    |   movel([0.479218, -1.510826, -2.472851, -0.728712, 1.570796, 2.050014],accel_mss,speed_ms,0,blend_radius_m)
    |   movel([0.479090, -1.510544, -2.473106, -0.728739, 1.570796, 2.049886],accel_mss,speed_ms,0,blend_radius_m)
    |   movel([0.478414, -1.510068, -2.473536, -0.728785, 1.570796, 2.049210],accel_mss,speed_ms,0,blend_radius_m)
    |   movel([0.477542, -1.509693, -2.473874, -0.728822, 1.570796, 2.048338],accel_mss,speed_ms,0,blend_radius_m)
    |   movel([0.475558, -1.508835, -2.474647, -0.728907, 1.570796, 2.046354],accel_mss,speed_ms,0,blend_radius_m)
    |   movel([0.473690, -1.507767, -2.475608, -0.729014, 1.570796, 2.044487],accel_mss,speed_ms,0,blend_radius_m)
    |   movel([0.472881, -1.507120, -2.476189, -0.729080, 1.570796, 2.043678],accel_mss,speed_ms,0,blend_radius_m)
    |   movel([0.472200, -1.506379, -2.476853, -0.729157, 1.570796, 2.042997],accel_mss,speed_ms,0,blend_radius_m)
    |   movel([0.471682, -1.505529, -2.477615, -0.729245, 1.570796, 2.042478],accel_mss,speed_ms,0,blend_radius_m)
    |   movel([0.471359, -1.504557, -2.478484, -0.729348, 1.570796, 2.042155],accel_mss,speed_ms,0,blend_radius_m)
    |   movel([0.472548, -1.505063, -2.478031, -0.729294, 1.570796, 2.043345],accel_mss,speed_ms,0,blend_radius_m)
    |   movel([0.473290, -1.505166, -2.477940, -0.729283, 1.570796, 2.044086],accel_mss,speed_ms,0,blend_radius_m)
    |   movel([0.473666, -1.505119, -2.477981, -0.729288, 1.570796, 2.044462],accel_mss,speed_ms,0,blend_radius_m)
    |   movel([0.474036, -1.504983, -2.478103, -0.729303, 1.570796, 2.044833],accel_mss,speed_ms,0,blend_radius_m)
    |   movel([0.474250, -1.504808, -2.478260, -0.729321, 1.570796, 2.045046],accel_mss,speed_ms,0,blend_radius_m)
    |   movel([0.474359, -1.504562, -2.478480, -0.729347, 1.570796, 2.045156],accel_mss,speed_ms,0,blend_radius_m)
    |   movel([0.474320, -1.503904, -2.479067, -0.729418, 1.570796, 2.045117],accel_mss,speed_ms,0,blend_radius_m)
    |   movel([0.474008, -1.503088, -2.479795, -0.729506, 1.570796, 2.044804],accel_mss,speed_ms,0,blend_radius_m)
    |   movel([0.473517, -1.502193, -2.480592, -0.729604, 1.570796, 2.044314],accel_mss,speed_ms,0,blend_radius_m)
    |   movel([0.471613, -1.499414, -2.483059, -0.729917, 1.570796, 2.042409],accel_mss,speed_ms,0,blend_radius_m)
    |   movel([0.471030, -1.498202, -2.484130, -0.730057, 1.570796, 2.041827],accel_mss,speed_ms,0,blend_radius_m)
    |   movel([0.470618, -1.496895, -2.485283, -0.730211, 1.570796, 2.041414],accel_mss,speed_ms,0,blend_radius_m)
    |   movel([0.470446, -1.495493, -2.486518, -0.730379, 1.570796, 2.041242],accel_mss,speed_ms,0,blend_radius_m)
    |   movel([0.470580, -1.493993, -2.487834, -0.730562, 1.570796, 2.041377],accel_mss,speed_ms,0,blend_radius_m)
    |   movel([0.471074, -1.495188, -2.486785, -0.730416, 1.570796, 2.041871],accel_mss,speed_ms,0,blend_radius_m)
    |   movel([0.471484, -1.495742, -2.486298, -0.730349, 1.570796, 2.042280],accel_mss,speed_ms,0,blend_radius_m)
    |   movel([0.472012, -1.496033, -2.486042, -0.730314, 1.570796, 2.042808],accel_mss,speed_ms,0,blend_radius_m)
    |   movel([0.472673, -1.496012, -2.486061, -0.730316, 1.570796, 2.043469],accel_mss,speed_ms,0,blend_radius_m)
    |   movel([0.473211, -1.495731, -2.486308, -0.730350, 1.570796, 2.044007],accel_mss,speed_ms,0,blend_radius_m)
    |   movel([0.473577, -1.495256, -2.486726, -0.730407, 1.570796, 2.044373],accel_mss,speed_ms,0,blend_radius_m)
    |   movel([0.473727, -1.494646, -2.487261, -0.730482, 1.570796, 2.044523],accel_mss,speed_ms,0,blend_radius_m)
    |   movel([0.473997, -1.491440, -2.490067, -0.730882, 1.570796, 2.044794],accel_mss,speed_ms,0,blend_radius_m)
    |   movel([0.474620, -1.488224, -2.492866, -0.731299, 1.570796, 2.045417],accel_mss,speed_ms,0,blend_radius_m)
    |   movel([0.475100, -1.486590, -2.494281, -0.731518, 1.570796, 2.045897],accel_mss,speed_ms,0,blend_radius_m)
    |   movel([0.475711, -1.484927, -2.495718, -0.731745, 1.570796, 2.046507],accel_mss,speed_ms,0,blend_radius_m)
    |   movel([0.476467, -1.483225, -2.497183, -0.731981, 1.570796, 2.047263],accel_mss,speed_ms,0,blend_radius_m)
    |   movel([0.477383, -1.481477, -2.498684, -0.732229, 1.570796, 2.048179],accel_mss,speed_ms,0,blend_radius_m)
    |   speed_ms = 0.005
    |   movel([0.477383, -1.473438, -2.495122, -0.743828, 1.570796, 2.048179],accel_mss,speed_ms,0,blend_radius_m)
    |   speed_ms = 0.040
    |   movel([0.466032, -1.452408, -2.512575, -0.747407, 1.570796, 2.036828],accel_mss,speed_ms,0,blend_radius_m)
    |   speed_ms = 0.005
    |   movel([0.466032, -1.460613, -2.516221, -0.735555, 1.570796, 2.036828],accel_mss,speed_ms,0,blend_radius_m)
    |   speed_ms = 0.025
    |   movel([0.468902, -1.458797, -2.517715, -0.735877, 1.570796, 2.039698],accel_mss,speed_ms,0,blend_radius_m)
    |   movel([0.471734, -1.456911, -2.519262, -0.736216, 1.570796, 2.042530],accel_mss,speed_ms,0,blend_radius_m)
    |   movel([0.477317, -1.452938, -2.522502, -0.736949, 1.570796, 2.048114],accel_mss,speed_ms,0,blend_radius_m)
    |   movel([0.482782, -1.448709, -2.525923, -0.737756, 1.570796, 2.053579],accel_mss,speed_ms,0,blend_radius_m)
    |   movel([0.488116, -1.444241, -2.529509, -0.738639, 1.570796, 2.058913],accel_mss,speed_ms,0,blend_radius_m)
    |   movel([0.493309, -1.439545, -2.533244, -0.739600, 1.570796, 2.064105],accel_mss,speed_ms,0,blend_radius_m)
    |   movel([0.498346, -1.434638, -2.537111, -0.740640, 1.570796, 2.069143],accel_mss,speed_ms,0,blend_radius_m)
    |   movel([0.503214, -1.429536, -2.541092, -0.741760, 1.570796, 2.074011],accel_mss,speed_ms,0,blend_radius_m)
    |   movel([0.507901, -1.424253, -2.545174, -0.742962, 1.570796, 2.078698],accel_mss,speed_ms,0,blend_radius_m)
    |   movel([0.512387, -1.418809, -2.549336, -0.744244, 1.570796, 2.083184],accel_mss,speed_ms,0,blend_radius_m)
    |   movel([0.516658, -1.413219, -2.553563, -0.745607, 1.570796, 2.087454],accel_mss,speed_ms,0,blend_radius_m)
    |   movel([0.520693, -1.407501, -2.557838, -0.747050, 1.570796, 2.091490],accel_mss,speed_ms,0,blend_radius_m)
    |   movel([0.524474, -1.401675, -2.562144, -0.748570, 1.570796, 2.095271],accel_mss,speed_ms,0,blend_radius_m)
    |   movel([0.527986, -1.395759, -2.566466, -0.750164, 1.570796, 2.098783],accel_mss,speed_ms,0,blend_radius_m)
    |   movel([0.531202, -1.389774, -2.570785, -0.751829, 1.570796, 2.101998],accel_mss,speed_ms,0,blend_radius_m)
    |   movel([0.534102, -1.383745, -2.575084, -0.753560, 1.570796, 2.104898],accel_mss,speed_ms,0,blend_radius_m)
    |   movel([0.537945, -1.374648, -2.581470, -0.756271, 1.570796, 2.108741],accel_mss,speed_ms,0,blend_radius_m)
    |   movel([0.538771, -1.373143, -2.582516, -0.756731, 1.570796, 2.109567],accel_mss,speed_ms,0,blend_radius_m)
    |   movel([0.539817, -1.371681, -2.583528, -0.757181, 1.570796, 2.110613],accel_mss,speed_ms,0,blend_radius_m)
    |   movel([0.541538, -1.369792, -2.584831, -0.757767, 1.570796, 2.112334],accel_mss,speed_ms,0,blend_radius_m)
    |   movel([0.543091, -1.368476, -2.585735, -0.758178, 1.570796, 2.113887],accel_mss,speed_ms,0,blend_radius_m)
    |   movel([0.543804, -1.368020, -2.586049, -0.758321, 1.570796, 2.114601],accel_mss,speed_ms,0,blend_radius_m)
    |   movel([0.545113, -1.367469, -2.586426, -0.758494, 1.570796, 2.115909],accel_mss,speed_ms,0,blend_radius_m)
    |   movel([0.545705, -1.367366, -2.586497, -0.758526, 1.570796, 2.116501],accel_mss,speed_ms,0,blend_radius_m)
    |   movel([0.546777, -1.367466, -2.586428, -0.758495, 1.570796, 2.117574],accel_mss,speed_ms,0,blend_radius_m)
    |   movel([0.547701, -1.367929, -2.586111, -0.758349, 1.570796, 2.118497],accel_mss,speed_ms,0,blend_radius_m)
    |   movel([0.548483, -1.368700, -2.585581, -0.758107, 1.570796, 2.119280],accel_mss,speed_ms,0,blend_radius_m)
    |   movel([0.549132, -1.369728, -2.584875, -0.757786, 1.570796, 2.119928],accel_mss,speed_ms,0,blend_radius_m)
    |   movel([0.549655, -1.370952, -2.584031, -0.757406, 1.570796, 2.120452],accel_mss,speed_ms,0,blend_radius_m)
    |   movel([0.550060, -1.372322, -2.583084, -0.756983, 1.570796, 2.120856],accel_mss,speed_ms,0,blend_radius_m)
    |   movel([0.550551, -1.375266, -2.581040, -0.756083, 1.570796, 2.121347],accel_mss,speed_ms,0,blend_radius_m)
    |   movel([0.550668, -1.378132, -2.579039, -0.755219, 1.570796, 2.121464],accel_mss,speed_ms,0,blend_radius_m)
    |   movel([0.550484, -1.380487, -2.577385, -0.754517, 1.570796, 2.121281],accel_mss,speed_ms,0,blend_radius_m)
    |   movel([0.549919, -1.383302, -2.575398, -0.753689, 1.570796, 2.120715],accel_mss,speed_ms,0,blend_radius_m)
    |   movel([0.549155, -1.386148, -2.573377, -0.752864, 1.570796, 2.119951],accel_mss,speed_ms,0,blend_radius_m)
    |   movel([0.547245, -1.391873, -2.569277, -0.751240, 1.570796, 2.118042],accel_mss,speed_ms,0,blend_radius_m)
    |   movel([0.545162, -1.397558, -2.565157, -0.749674, 1.570796, 2.115959],accel_mss,speed_ms,0,blend_radius_m)
    |   movel([0.543302, -1.403099, -2.561096, -0.748194, 1.570796, 2.114098],accel_mss,speed_ms,0,blend_radius_m)
    |   movel([0.541964, -1.407989, -2.557475, -0.746925, 1.570796, 2.112760],accel_mss,speed_ms,0,blend_radius_m)
    |   movel([0.541538, -1.410366, -2.555702, -0.746321, 1.570796, 2.112334],accel_mss,speed_ms,0,blend_radius_m)
    |   movel([0.541409, -1.412652, -2.553988, -0.745748, 1.570796, 2.112205],accel_mss,speed_ms,0,blend_radius_m)
    |   movel([0.541530, -1.413653, -2.553236, -0.745500, 1.570796, 2.112327],accel_mss,speed_ms,0,blend_radius_m)
    |   movel([0.541712, -1.414085, -2.552911, -0.745393, 1.570796, 2.112508],accel_mss,speed_ms,0,blend_radius_m)
    |   movel([0.542014, -1.414430, -2.552651, -0.745308, 1.570796, 2.112811],accel_mss,speed_ms,0,blend_radius_m)
    |   movel([0.542579, -1.414692, -2.552453, -0.745244, 1.570796, 2.113375],accel_mss,speed_ms,0,blend_radius_m)
    |   movel([0.543278, -1.414768, -2.552396, -0.745225, 1.570796, 2.114074],accel_mss,speed_ms,0,blend_radius_m)
    |   movel([0.544866, -1.414552, -2.552559, -0.745278, 1.570796, 2.115662],accel_mss,speed_ms,0,blend_radius_m)
    |   movel([0.546735, -1.414053, -2.552935, -0.745401, 1.570796, 2.117531],accel_mss,speed_ms,0,blend_radius_m)
    |   movel([0.548597, -1.413416, -2.553414, -0.745558, 1.570796, 2.119394],accel_mss,speed_ms,0,blend_radius_m)
    |   movel([0.552310, -1.411832, -2.554605, -0.745953, 1.570796, 2.123106],accel_mss,speed_ms,0,blend_radius_m)
    |   movel([0.559726, -1.408243, -2.557286, -0.746860, 1.570796, 2.130523],accel_mss,speed_ms,0,blend_radius_m)
    |   movel([0.563228, -1.406710, -2.558426, -0.747253, 1.570796, 2.134025],accel_mss,speed_ms,0,blend_radius_m)
    |   movel([0.565185, -1.405992, -2.558959, -0.747439, 1.570796, 2.135981],accel_mss,speed_ms,0,blend_radius_m)
    |   movel([0.567041, -1.405492, -2.559329, -0.747568, 1.570796, 2.137837],accel_mss,speed_ms,0,blend_radius_m)
    |   movel([0.567877, -1.405366, -2.559422, -0.747601, 1.570796, 2.138673],accel_mss,speed_ms,0,blend_radius_m)
    |   movel([0.568623, -1.405347, -2.559436, -0.747606, 1.570796, 2.139419],accel_mss,speed_ms,0,blend_radius_m)
    |   movel([0.569256, -1.405450, -2.559360, -0.747579, 1.570796, 2.140052],accel_mss,speed_ms,0,blend_radius_m)
    |   movel([0.569753, -1.405695, -2.559178, -0.747516, 1.570796, 2.140549],accel_mss,speed_ms,0,blend_radius_m)
    |   movel([0.570094, -1.406095, -2.558882, -0.747412, 1.570796, 2.140890],accel_mss,speed_ms,0,blend_radius_m)
    |   movel([0.570258, -1.406668, -2.558457, -0.747264, 1.570796, 2.141054],accel_mss,speed_ms,0,blend_radius_m)
    |   movel([0.570222, -1.407432, -2.557890, -0.747068, 1.570796, 2.141018],accel_mss,speed_ms,0,blend_radius_m)
    |   movel([0.569963, -1.408401, -2.557168, -0.746820, 1.570796, 2.140760],accel_mss,speed_ms,0,blend_radius_m)
    |   movel([0.569286, -1.410124, -2.555883, -0.746382, 1.570796, 2.140083],accel_mss,speed_ms,0,blend_radius_m)
    |   movel([0.568475, -1.411800, -2.554629, -0.745961, 1.570796, 2.139271],accel_mss,speed_ms,0,blend_radius_m)
    |   movel([0.567540, -1.413425, -2.553408, -0.745556, 1.570796, 2.138336],accel_mss,speed_ms,0,blend_radius_m)
    |   movel([0.566489, -1.415003, -2.552219, -0.745167, 1.570796, 2.137285],accel_mss,speed_ms,0,blend_radius_m)
    |   movel([0.565332, -1.416528, -2.551066, -0.744795, 1.570796, 2.136128],accel_mss,speed_ms,0,blend_radius_m)
    |   movel([0.564077, -1.418002, -2.549949, -0.744438, 1.570796, 2.134873],accel_mss,speed_ms,0,blend_radius_m)
    |   movel([0.562731, -1.419423, -2.548869, -0.744097, 1.570796, 2.133528],accel_mss,speed_ms,0,blend_radius_m)
    |   movel([0.561305, -1.420792, -2.547825, -0.743772, 1.570796, 2.132101],accel_mss,speed_ms,0,blend_radius_m)
    |   movel([0.558245, -1.423366, -2.545855, -0.743168, 1.570796, 2.129041],accel_mss,speed_ms,0,blend_radius_m)
    |   movel([0.554959, -1.425720, -2.544045, -0.742624, 1.570796, 2.125756],accel_mss,speed_ms,0,blend_radius_m)
    |   movel([0.551512, -1.427846, -2.542403, -0.742140, 1.570796, 2.122308],accel_mss,speed_ms,0,blend_radius_m)
    |   movel([0.547970, -1.429739, -2.540935, -0.741715, 1.570796, 2.118766],accel_mss,speed_ms,0,blend_radius_m)
    |   movel([0.539979, -1.433664, -2.537874, -0.740851, 1.570796, 2.110775],accel_mss,speed_ms,0,blend_radius_m)
    |   movel([0.535909, -1.435398, -2.536514, -0.740477, 1.570796, 2.106705],accel_mss,speed_ms,0,blend_radius_m)
    |   movel([0.533914, -1.436111, -2.535954, -0.740324, 1.570796, 2.104710],accel_mss,speed_ms,0,blend_radius_m)
    |   movel([0.531965, -1.436684, -2.535503, -0.740202, 1.570796, 2.102762],accel_mss,speed_ms,0,blend_radius_m)
    |   movel([0.530749, -1.436952, -2.535292, -0.740145, 1.570796, 2.101545],accel_mss,speed_ms,0,blend_radius_m)
    |   movel([0.529585, -1.437111, -2.535167, -0.740111, 1.570796, 2.100382],accel_mss,speed_ms,0,blend_radius_m)
    |   movel([0.528488, -1.437147, -2.535138, -0.740104, 1.570796, 2.099284],accel_mss,speed_ms,0,blend_radius_m)
    |   movel([0.527472, -1.437051, -2.535214, -0.740124, 1.570796, 2.098268],accel_mss,speed_ms,0,blend_radius_m)
    |   movel([0.526552, -1.436813, -2.535401, -0.740174, 1.570796, 2.097349],accel_mss,speed_ms,0,blend_radius_m)
    |   movel([0.525742, -1.436422, -2.535709, -0.740258, 1.570796, 2.096539],accel_mss,speed_ms,0,blend_radius_m)
    |   movel([0.525060, -1.435863, -2.536149, -0.740377, 1.570796, 2.095857],accel_mss,speed_ms,0,blend_radius_m)
    |   movel([0.524520, -1.435125, -2.536729, -0.740535, 1.570796, 2.095316],accel_mss,speed_ms,0,blend_radius_m)
    |   movel([0.524155, -1.434223, -2.537437, -0.740730, 1.570796, 2.094952],accel_mss,speed_ms,0,blend_radius_m)
    |   movel([0.523975, -1.433243, -2.538203, -0.740942, 1.570796, 2.094772],accel_mss,speed_ms,0,blend_radius_m)
    |   movel([0.523875, -1.429029, -2.541486, -0.741874, 1.570796, 2.094671],accel_mss,speed_ms,0,blend_radius_m)
    |   movel([0.523695, -1.428021, -2.542268, -0.742101, 1.570796, 2.094491],accel_mss,speed_ms,0,blend_radius_m)
    |   movel([0.523325, -1.427082, -2.542994, -0.742313, 1.570796, 2.094122],accel_mss,speed_ms,0,blend_radius_m)
    |   movel([0.523071, -1.426813, -2.543202, -0.742374, 1.570796, 2.093867],accel_mss,speed_ms,0,blend_radius_m)
    |   movel([0.522822, -1.426930, -2.543111, -0.742348, 1.570796, 2.093618],accel_mss,speed_ms,0,blend_radius_m)
    |   movel([0.522355, -1.427345, -2.542790, -0.742254, 1.570796, 2.093151],accel_mss,speed_ms,0,blend_radius_m)
    |   movel([0.520874, -1.428916, -2.541574, -0.741899, 1.570796, 2.091670],accel_mss,speed_ms,0,blend_radius_m)
    |   movel([0.516616, -1.433877, -2.537707, -0.740805, 1.570796, 2.087413],accel_mss,speed_ms,0,blend_radius_m)
    |   movel([0.509629, -1.442253, -2.531094, -0.739042, 1.570796, 2.080425],accel_mss,speed_ms,0,blend_radius_m)
    |   movel([0.505584, -1.446410, -2.527772, -0.738207, 1.570796, 2.076380],accel_mss,speed_ms,0,blend_radius_m)
    |   movel([0.501403, -1.450431, -2.524534, -0.737424, 1.570796, 2.072199],accel_mss,speed_ms,0,blend_radius_m)
    |   movel([0.497105, -1.454321, -2.521377, -0.736691, 1.570796, 2.067901],accel_mss,speed_ms,0,blend_radius_m)
    |   movel([0.492719, -1.458086, -2.518299, -0.736004, 1.570796, 2.063515],accel_mss,speed_ms,0,blend_radius_m)
    |   movel([0.487033, -1.462788, -2.514425, -0.735177, 1.570796, 2.057830],accel_mss,speed_ms,0,blend_radius_m)
    |   movel([0.481276, -1.467394, -2.510596, -0.734399, 1.570796, 2.052072],accel_mss,speed_ms,0,blend_radius_m)
    |   movel([0.475444, -1.471860, -2.506851, -0.733677, 1.570796, 2.046241],accel_mss,speed_ms,0,blend_radius_m)
    |   movel([0.469530, -1.476139, -2.503235, -0.733015, 1.570796, 2.040326],accel_mss,speed_ms,0,blend_radius_m)
    |   movel([0.463529, -1.480182, -2.499792, -0.732415, 1.570796, 2.034326],accel_mss,speed_ms,0,blend_radius_m)
    |   movel([0.460496, -1.482104, -2.498146, -0.732139, 1.570796, 2.031292],accel_mss,speed_ms,0,blend_radius_m)
    |   movel([0.457435, -1.483950, -2.496559, -0.731880, 1.570796, 2.028231],accel_mss,speed_ms,0,blend_radius_m)
    |   movel([0.454348, -1.485717, -2.495035, -0.731636, 1.570796, 2.025144],accel_mss,speed_ms,0,blend_radius_m)
    |   movel([0.451235, -1.487398, -2.493582, -0.731409, 1.570796, 2.022032],accel_mss,speed_ms,0,blend_radius_m)
    |   movel([0.448093, -1.488991, -2.492200, -0.731198, 1.570796, 2.018889],accel_mss,speed_ms,0,blend_radius_m)
    |   movel([0.444920, -1.490485, -2.490900, -0.731004, 1.570796, 2.015717],accel_mss,speed_ms,0,blend_radius_m)
    |   movel([0.441121, -1.492138, -2.489458, -0.730793, 1.570796, 2.011917],accel_mss,speed_ms,0,blend_radius_m)
    |   movel([0.439214, -1.492856, -2.488830, -0.730703, 1.570796, 2.010010],accel_mss,speed_ms,0,blend_radius_m)
    |   movel([0.435953, -1.493815, -2.487990, -0.730584, 1.570796, 2.006750],accel_mss,speed_ms,0,blend_radius_m)
    |   movel([0.434355, -1.494140, -2.487706, -0.730544, 1.570796, 2.005151],accel_mss,speed_ms,0,blend_radius_m)
    |   movel([0.432892, -1.494199, -2.487654, -0.730536, 1.570796, 2.003689],accel_mss,speed_ms,0,blend_radius_m)
    |   movel([0.432332, -1.494057, -2.487778, -0.730554, 1.570796, 2.003129],accel_mss,speed_ms,0,blend_radius_m)
    |   movel([0.431947, -1.493762, -2.488037, -0.730590, 1.570796, 2.002743],accel_mss,speed_ms,0,blend_radius_m)
    |   movel([0.433050, -1.492467, -2.489170, -0.730752, 1.570796, 2.003846],accel_mss,speed_ms,0,blend_radius_m)
    |   movel([0.433977, -1.491111, -2.490354, -0.730924, 1.570796, 2.004774],accel_mss,speed_ms,0,blend_radius_m)
    |   movel([0.434304, -1.490444, -2.490936, -0.731009, 1.570796, 2.005100],accel_mss,speed_ms,0,blend_radius_m)
    |   movel([0.434501, -1.489802, -2.491495, -0.731092, 1.570796, 2.005297],accel_mss,speed_ms,0,blend_radius_m)
    |   movel([0.434541, -1.489197, -2.492021, -0.731171, 1.570796, 2.005338],accel_mss,speed_ms,0,blend_radius_m)
    |   movel([0.434390, -1.488645, -2.492501, -0.731244, 1.570796, 2.005186],accel_mss,speed_ms,0,blend_radius_m)
    |   movel([0.433605, -1.487527, -2.493470, -0.731392, 1.570796, 2.004401],accel_mss,speed_ms,0,blend_radius_m)
    |   movel([0.433481, -1.487048, -2.493885, -0.731456, 1.570796, 2.004278],accel_mss,speed_ms,0,blend_radius_m)
    |   movel([0.433504, -1.486523, -2.494339, -0.731527, 1.570796, 2.004300],accel_mss,speed_ms,0,blend_radius_m)
    |   movel([0.433910, -1.485389, -2.495318, -0.731681, 1.570796, 2.004706],accel_mss,speed_ms,0,blend_radius_m)
    |   movel([0.434649, -1.484208, -2.496337, -0.731844, 1.570796, 2.005445],accel_mss,speed_ms,0,blend_radius_m)
    |   movel([0.435548, -1.483069, -2.497317, -0.732003, 1.570796, 2.006344],accel_mss,speed_ms,0,blend_radius_m)
    |   movel([0.438447, -1.479730, -2.500178, -0.732481, 1.570796, 2.009243],accel_mss,speed_ms,0,blend_radius_m)
    |   movel([0.441555, -1.476440, -2.502980, -0.732969, 1.570796, 2.012351],accel_mss,speed_ms,0,blend_radius_m)
    |   movel([0.443204, -1.474853, -2.504325, -0.733211, 1.570796, 2.014000],accel_mss,speed_ms,0,blend_radius_m)
    |   movel([0.444924, -1.473320, -2.505621, -0.733448, 1.570796, 2.015721],accel_mss,speed_ms,0,blend_radius_m)
    |   movel([0.446722, -1.471861, -2.506851, -0.733677, 1.570796, 2.017518],accel_mss,speed_ms,0,blend_radius_m)
    |   movel([0.448605, -1.470491, -2.508003, -0.733895, 1.570796, 2.019402],accel_mss,speed_ms,0,blend_radius_m)
    |   movel([0.450533, -1.469313, -2.508991, -0.734085, 1.570796, 2.021329],accel_mss,speed_ms,0,blend_radius_m)
    |   movel([0.456408, -1.466369, -2.511451, -0.734569, 1.570796, 2.027205],accel_mss,speed_ms,0,blend_radius_m)
    |   movel([0.461233, -1.463560, -2.513785, -0.735044, 1.570796, 2.032030],accel_mss,speed_ms,0,blend_radius_m)
    |   movel([0.466032, -1.460613, -2.516221, -0.735555, 1.570796, 2.036828],accel_mss,speed_ms,0,blend_radius_m)
    |   movel([0.468181, -1.459252, -2.517341, -0.735796, 1.570796, 2.038977],accel_mss,speed_ms,0,blend_radius_m)
    |   speed_ms = 0.005
    |   movel([0.468181, -1.451036, -2.513689, -0.747664, 1.570796, 2.038977],accel_mss,speed_ms,0,blend_radius_m)
    |   speed_ms = 0.040
    |   movel([0.426259, -1.473575, -2.495006, -0.743807, 1.570796, 1.997056],accel_mss,speed_ms,0,blend_radius_m)
    |   speed_ms = 0.005
    |   movel([0.426259, -1.481613, -2.498567, -0.732209, 1.570796, 1.997056],accel_mss,speed_ms,0,blend_radius_m)
    |   speed_ms = 0.025
    |   movel([0.426785, -1.485296, -2.495399, -0.731694, 1.570796, 1.997582],accel_mss,speed_ms,0,blend_radius_m)
    |   movel([0.426943, -1.487302, -2.493665, -0.731422, 1.570796, 1.997739],accel_mss,speed_ms,0,blend_radius_m)
    |   movel([0.426956, -1.489374, -2.491867, -0.731148, 1.570796, 1.997753],accel_mss,speed_ms,0,blend_radius_m)
    |   movel([0.426780, -1.491475, -2.490037, -0.730877, 1.570796, 1.997576],accel_mss,speed_ms,0,blend_radius_m)
    |   movel([0.426361, -1.493570, -2.488205, -0.730614, 1.570796, 1.997157],accel_mss,speed_ms,0,blend_radius_m)
    |   movel([0.425648, -1.495628, -2.486399, -0.730362, 1.570796, 1.996444],accel_mss,speed_ms,0,blend_radius_m)
    |   movel([0.425164, -1.496634, -2.485513, -0.730242, 1.570796, 1.995961],accel_mss,speed_ms,0,blend_radius_m)
    |   movel([0.424590, -1.497615, -2.484648, -0.730126, 1.570796, 1.995386],accel_mss,speed_ms,0,blend_radius_m)
    |   movel([0.424302, -1.496994, -2.485196, -0.730199, 1.570796, 1.995098],accel_mss,speed_ms,0,blend_radius_m)
    |   movel([0.424245, -1.496354, -2.485760, -0.730275, 1.570796, 1.995041],accel_mss,speed_ms,0,blend_radius_m)
    |   movel([0.424185, -1.494900, -2.487039, -0.730451, 1.570796, 1.994982],accel_mss,speed_ms,0,blend_radius_m)
    |   movel([0.423788, -1.493467, -2.488295, -0.730627, 1.570796, 1.994585],accel_mss,speed_ms,0,blend_radius_m)
    |   movel([0.423223, -1.492114, -2.489479, -0.730796, 1.570796, 1.994019],accel_mss,speed_ms,0,blend_radius_m)
    |   movel([0.422503, -1.490843, -2.490588, -0.730958, 1.570796, 1.993300],accel_mss,speed_ms,0,blend_radius_m)
    |   movel([0.421640, -1.489659, -2.491619, -0.731111, 1.570796, 1.992436],accel_mss,speed_ms,0,blend_radius_m)
    |   movel([0.420645, -1.488568, -2.492567, -0.731254, 1.570796, 1.991442],accel_mss,speed_ms,0,blend_radius_m)
    |   movel([0.419531, -1.487577, -2.493427, -0.731385, 1.570796, 1.990327],accel_mss,speed_ms,0,blend_radius_m)
    |   movel([0.418306, -1.486690, -2.494195, -0.731504, 1.570796, 1.989103],accel_mss,speed_ms,0,blend_radius_m)
    |   movel([0.416988, -1.485911, -2.494868, -0.731610, 1.570796, 1.987784],accel_mss,speed_ms,0,blend_radius_m)
    |   movel([0.416041, -1.485484, -2.495237, -0.731668, 1.570796, 1.986838],accel_mss,speed_ms,0,blend_radius_m)
    |   movel([0.415222, -1.485270, -2.495421, -0.731697, 1.570796, 1.986019],accel_mss,speed_ms,0,blend_radius_m)
    |   movel([0.414524, -1.485248, -2.495440, -0.731700, 1.570796, 1.985320],accel_mss,speed_ms,0,blend_radius_m)
    |   movel([0.413938, -1.485397, -2.495312, -0.731680, 1.570796, 1.984734],accel_mss,speed_ms,0,blend_radius_m)
    |   movel([0.413451, -1.485701, -2.495049, -0.731638, 1.570796, 1.984247],accel_mss,speed_ms,0,blend_radius_m)
    |   movel([0.413056, -1.486139, -2.494671, -0.731579, 1.570796, 1.983852],accel_mss,speed_ms,0,blend_radius_m)
    |   movel([0.412740, -1.486691, -2.494194, -0.731504, 1.570796, 1.983536],accel_mss,speed_ms,0,blend_radius_m)
    |   movel([0.412496, -1.487338, -2.493634, -0.731417, 1.570796, 1.983292],accel_mss,speed_ms,0,blend_radius_m)
    |   movel([0.412176, -1.488839, -2.492331, -0.731218, 1.570796, 1.982973],accel_mss,speed_ms,0,blend_radius_m)
    |   movel([0.411827, -1.493652, -2.488133, -0.730604, 1.570796, 1.982623],accel_mss,speed_ms,0,blend_radius_m)
    |   movel([0.411194, -1.492016, -2.489564, -0.730809, 1.570796, 1.981990],accel_mss,speed_ms,0,blend_radius_m)
    |   movel([0.410024, -1.488695, -2.492457, -0.731237, 1.570796, 1.980820],accel_mss,speed_ms,0,blend_radius_m)
    |   movel([0.409157, -1.487197, -2.493756, -0.731436, 1.570796, 1.979953],accel_mss,speed_ms,0,blend_radius_m)
    |   movel([0.407933, -1.485717, -2.495036, -0.731636, 1.570796, 1.978730],accel_mss,speed_ms,0,blend_radius_m)
    |   movel([0.406592, -1.484312, -2.496248, -0.731830, 1.570796, 1.977388],accel_mss,speed_ms,0,blend_radius_m)
    |   movel([0.403823, -1.481556, -2.498615, -0.732217, 1.570796, 1.974619],accel_mss,speed_ms,0,blend_radius_m)
    |   movel([0.402529, -1.480121, -2.499844, -0.732424, 1.570796, 1.973326],accel_mss,speed_ms,0,blend_radius_m)
    |   movel([0.401388, -1.478591, -2.501149, -0.732648, 1.570796, 1.972184],accel_mss,speed_ms,0,blend_radius_m)
    |   movel([0.400466, -1.476926, -2.502567, -0.732896, 1.570796, 1.971262],accel_mss,speed_ms,0,blend_radius_m)
    |   movel([0.399832, -1.475077, -2.504136, -0.733177, 1.570796, 1.970629],accel_mss,speed_ms,0,blend_radius_m)
    |   movel([0.399145, -1.479131, -2.500689, -0.732569, 1.570796, 1.969941],accel_mss,speed_ms,0,blend_radius_m)
    |   movel([0.398904, -1.481187, -2.498932, -0.732270, 1.570796, 1.969701],accel_mss,speed_ms,0,blend_radius_m)
    |   movel([0.398906, -1.483032, -2.497348, -0.732008, 1.570796, 1.969703],accel_mss,speed_ms,0,blend_radius_m)
    |   movel([0.398200, -1.481266, -2.498864, -0.732259, 1.570796, 1.968996],accel_mss,speed_ms,0,blend_radius_m)
    |   movel([0.397271, -1.479624, -2.500269, -0.732497, 1.570796, 1.968068],accel_mss,speed_ms,0,blend_radius_m)
    |   movel([0.395194, -1.476458, -2.502964, -0.732967, 1.570796, 1.965991],accel_mss,speed_ms,0,blend_radius_m)
    |   movel([0.394608, -1.475326, -2.503925, -0.733139, 1.570796, 1.965405],accel_mss,speed_ms,0,blend_radius_m)
    |   movel([0.394185, -1.474140, -2.504928, -0.733321, 1.570796, 1.964981],accel_mss,speed_ms,0,blend_radius_m)
    |   movel([0.393661, -1.471651, -2.507028, -0.733710, 1.570796, 1.964457],accel_mss,speed_ms,0,blend_radius_m)
    |   movel([0.393279, -1.469083, -2.509184, -0.734123, 1.570796, 1.964076],accel_mss,speed_ms,0,blend_radius_m)
    |   movel([0.392690, -1.466536, -2.511311, -0.734542, 1.570796, 1.963486],accel_mss,speed_ms,0,blend_radius_m)
    |   movel([0.392390, -1.465786, -2.511936, -0.734667, 1.570796, 1.963186],accel_mss,speed_ms,0,blend_radius_m)
    |   movel([0.391952, -1.465122, -2.512488, -0.734778, 1.570796, 1.962748],accel_mss,speed_ms,0,blend_radius_m)
    |   movel([0.391326, -1.464651, -2.512880, -0.734858, 1.570796, 1.962122],accel_mss,speed_ms,0,blend_radius_m)
    |   movel([0.390931, -1.464520, -2.512989, -0.734880, 1.570796, 1.961727],accel_mss,speed_ms,0,blend_radius_m)
    |   movel([0.390469, -1.464478, -2.513023, -0.734887, 1.570796, 1.961266],accel_mss,speed_ms,0,blend_radius_m)
    |   movel([0.389918, -1.464541, -2.512972, -0.734877, 1.570796, 1.960714],accel_mss,speed_ms,0,blend_radius_m)
    |   movel([0.389364, -1.464708, -2.512833, -0.734849, 1.570796, 1.960160],accel_mss,speed_ms,0,blend_radius_m)
    |   movel([0.388261, -1.465288, -2.512351, -0.734751, 1.570796, 1.959057],accel_mss,speed_ms,0,blend_radius_m)
    |   movel([0.387204, -1.466087, -2.511686, -0.734616, 1.570796, 1.958001],accel_mss,speed_ms,0,blend_radius_m)
    |   movel([0.386238, -1.466975, -2.510946, -0.734469, 1.570796, 1.957034],accel_mss,speed_ms,0,blend_radius_m)
    |   movel([0.386761, -1.465043, -2.512554, -0.734792, 1.570796, 1.957557],accel_mss,speed_ms,0,blend_radius_m)
    |   movel([0.387114, -1.463166, -2.514112, -0.735111, 1.570796, 1.957911],accel_mss,speed_ms,0,blend_radius_m)
    |   movel([0.387493, -1.459519, -2.517122, -0.735748, 1.570796, 1.958289],accel_mss,speed_ms,0,blend_radius_m)
    |   movel([0.387757, -1.455899, -2.520090, -0.736401, 1.570796, 1.958553],accel_mss,speed_ms,0,blend_radius_m)
    |   movel([0.388297, -1.452167, -2.523127, -0.737094, 1.570796, 1.959094],accel_mss,speed_ms,0,blend_radius_m)
    |   movel([0.388714, -1.450679, -2.524333, -0.737377, 1.570796, 1.959510],accel_mss,speed_ms,0,blend_radius_m)
    |   movel([0.389333, -1.449137, -2.525579, -0.737674, 1.570796, 1.960129],accel_mss,speed_ms,0,blend_radius_m)
    |   movel([0.390119, -1.447559, -2.526849, -0.737981, 1.570796, 1.960915],accel_mss,speed_ms,0,blend_radius_m)
    |   movel([0.391033, -1.445967, -2.528127, -0.738295, 1.570796, 1.961829],accel_mss,speed_ms,0,blend_radius_m)
    |   movel([0.393120, -1.442815, -2.530647, -0.738927, 1.570796, 1.963916],accel_mss,speed_ms,0,blend_radius_m)
    |   movel([0.395304, -1.439843, -2.533008, -0.739538, 1.570796, 1.966100],accel_mss,speed_ms,0,blend_radius_m)
    |   speed_ms = 0.005
    |   movel([0.395304, -1.431474, -2.529275, -0.751640, 1.570796, 1.966100],accel_mss,speed_ms,0,blend_radius_m)
    |   speed_ms = 0.040
    |   # Splitting Linear movement in 2 (instruction 806: MoveL 765)
    |   movel([0.433547, -1.397430, -2.555032, -0.759927, 1.570796, 2.004344],accel_mss,speed_ms,0,blend_radius_m)
    |   movel([0.474434, -1.362082, -2.579990, -0.770317, 1.570796, 2.045231],accel_mss,speed_ms,0,blend_radius_m)
    |   speed_ms = 0.005
    |   movel([0.474434, -1.370965, -2.584022, -0.757402, 1.570796, 2.045231],accel_mss,speed_ms,0,blend_radius_m)
    |   speed_ms = 0.025
    |   movel([0.472989, -1.371456, -2.583683, -0.757250, 1.570796, 2.043785],accel_mss,speed_ms,0,blend_radius_m)
    |   movel([0.472799, -1.371633, -2.583560, -0.757195, 1.570796, 2.043595],accel_mss,speed_ms,0,blend_radius_m)
    |   movel([0.472675, -1.372000, -2.583307, -0.757082, 1.570796, 2.043471],accel_mss,speed_ms,0,blend_radius_m)
    |   movel([0.472603, -1.373262, -2.582433, -0.756694, 1.570796, 2.043400],accel_mss,speed_ms,0,blend_radius_m)
    |   movel([0.473061, -1.377529, -2.579460, -0.755399, 1.570796, 2.043857],accel_mss,speed_ms,0,blend_radius_m)
    |   movel([0.474120, -1.383440, -2.575300, -0.753649, 1.570796, 2.044916],accel_mss,speed_ms,0,blend_radius_m)
    |   movel([0.475543, -1.390187, -2.570489, -0.751713, 1.570796, 2.046339],accel_mss,speed_ms,0,blend_radius_m)
    |   movel([0.478558, -1.403067, -2.561120, -0.748202, 1.570796, 2.049354],accel_mss,speed_ms,0,blend_radius_m)
    |   movel([0.480397, -1.410133, -2.555876, -0.746380, 1.570796, 2.051193],accel_mss,speed_ms,0,blend_radius_m)
    |   movel([0.480639, -1.410710, -2.555445, -0.746234, 1.570796, 2.051436],accel_mss,speed_ms,0,blend_radius_m)
    |   movel([0.481007, -1.411202, -2.555076, -0.746111, 1.570796, 2.051803],accel_mss,speed_ms,0,blend_radius_m)
    |   movel([0.481528, -1.411486, -2.554864, -0.746039, 1.570796, 2.052324],accel_mss,speed_ms,0,blend_radius_m)
    |   movel([0.481855, -1.411515, -2.554842, -0.746032, 1.570796, 2.052651],accel_mss,speed_ms,0,blend_radius_m)
    |   movel([0.482232, -1.411444, -2.554895, -0.746050, 1.570796, 2.053028],accel_mss,speed_ms,0,blend_radius_m)
    |   movel([0.482920, -1.411095, -2.555156, -0.746137, 1.570796, 2.053716],accel_mss,speed_ms,0,blend_radius_m)
    |   movel([0.483556, -1.410598, -2.555529, -0.746263, 1.570796, 2.054352],accel_mss,speed_ms,0,blend_radius_m)
    |   movel([0.486901, -1.407573, -2.557785, -0.747032, 1.570796, 2.057697],accel_mss,speed_ms,0,blend_radius_m)
    |   movel([0.490066, -1.404379, -2.560152, -0.747858, 1.570796, 2.060862],accel_mss,speed_ms,0,blend_radius_m)
    |   movel([0.493048, -1.401044, -2.562608, -0.748737, 1.570796, 2.063844],accel_mss,speed_ms,0,blend_radius_m)
    |   movel([0.495856, -1.397597, -2.565129, -0.749663, 1.570796, 2.066652],accel_mss,speed_ms,0,blend_radius_m)
    |   movel([0.498491, -1.394061, -2.567697, -0.750631, 1.570796, 2.069287],accel_mss,speed_ms,0,blend_radius_m)
    |   movel([0.500957, -1.390465, -2.570289, -0.751635, 1.570796, 2.071754],accel_mss,speed_ms,0,blend_radius_m)
    |   movel([0.503258, -1.386836, -2.572887, -0.752666, 1.570796, 2.074055],accel_mss,speed_ms,0,blend_radius_m)
    |   movel([0.505395, -1.383207, -2.575465, -0.753717, 1.570796, 2.076191],accel_mss,speed_ms,0,blend_radius_m)
    |   movel([0.506270, -1.381540, -2.576643, -0.754206, 1.570796, 2.077066],accel_mss,speed_ms,0,blend_radius_m)
    |   movel([0.506956, -1.379963, -2.577753, -0.754673, 1.570796, 2.077752],accel_mss,speed_ms,0,blend_radius_m)
    |   movel([0.507455, -1.378474, -2.578799, -0.755116, 1.570796, 2.078251],accel_mss,speed_ms,0,blend_radius_m)
    |   movel([0.507775, -1.377073, -2.579780, -0.755537, 1.570796, 2.078572],accel_mss,speed_ms,0,blend_radius_m)
    |   movel([0.507919, -1.375760, -2.580696, -0.755933, 1.570796, 2.078715],accel_mss,speed_ms,0,blend_radius_m)
    |   movel([0.507889, -1.374537, -2.581547, -0.756305, 1.570796, 2.078686],accel_mss,speed_ms,0,blend_radius_m)
    |   movel([0.507696, -1.373399, -2.582338, -0.756652, 1.570796, 2.078492],accel_mss,speed_ms,0,blend_radius_m)
    |   movel([0.507340, -1.372345, -2.583068, -0.756976, 1.570796, 2.078137],accel_mss,speed_ms,0,blend_radius_m)
    |   movel([0.506829, -1.371378, -2.583737, -0.757274, 1.570796, 2.077625],accel_mss,speed_ms,0,blend_radius_m)
    |   movel([0.506167, -1.370497, -2.584345, -0.757547, 1.570796, 2.076963],accel_mss,speed_ms,0,blend_radius_m)
    |   movel([0.505358, -1.369697, -2.584896, -0.757796, 1.570796, 2.076154],accel_mss,speed_ms,0,blend_radius_m)
    |   movel([0.504410, -1.368982, -2.585388, -0.758019, 1.570796, 2.075207],accel_mss,speed_ms,0,blend_radius_m)
    |   movel([0.502113, -1.367799, -2.586200, -0.758390, 1.570796, 2.072910],accel_mss,speed_ms,0,blend_radius_m)
    |   movel([0.499324, -1.366940, -2.586788, -0.758661, 1.570796, 2.070120],accel_mss,speed_ms,0,blend_radius_m)
    |   movel([0.496587, -1.366526, -2.587072, -0.758791, 1.570796, 2.067383],accel_mss,speed_ms,0,blend_radius_m)
    |   movel([0.493687, -1.366467, -2.587112, -0.758810, 1.570796, 2.064483],accel_mss,speed_ms,0,blend_radius_m)
    |   movel([0.490645, -1.366722, -2.586938, -0.758729, 1.570796, 2.061441],accel_mss,speed_ms,0,blend_radius_m)
    |   movel([0.487496, -1.367238, -2.586584, -0.758567, 1.570796, 2.058292],accel_mss,speed_ms,0,blend_radius_m)
    |   movel([0.484273, -1.367969, -2.586083, -0.758337, 1.570796, 2.055069],accel_mss,speed_ms,0,blend_radius_m)
    |   movel([0.481001, -1.368865, -2.585468, -0.758056, 1.570796, 2.051797],accel_mss,speed_ms,0,blend_radius_m)
    |   movel([0.474434, -1.370965, -2.584022, -0.757402, 1.570796, 2.045231],accel_mss,speed_ms,0,blend_radius_m)
    |   movel([0.472989, -1.371456, -2.583683, -0.757250, 1.570796, 2.043785],accel_mss,speed_ms,0,blend_radius_m)
    |   movel([0.472799, -1.371633, -2.583560, -0.757195, 1.570796, 2.043595],accel_mss,speed_ms,0,blend_radius_m)
    |   movel([0.472675, -1.372000, -2.583307, -0.757082, 1.570796, 2.043471],accel_mss,speed_ms,0,blend_radius_m)
    |   movel([0.472651, -1.372400, -2.583030, -0.756959, 1.570796, 2.043448],accel_mss,speed_ms,0,blend_radius_m)
    |   speed_ms = 0.005
    |   movel([0.472651, -1.363527, -2.579005, -0.769857, 1.570796, 2.043448],accel_mss,speed_ms,0,blend_radius_m)
    |   speed_ms = 0.040
    |   movel([0.476821, -1.340541, -2.594336, -0.777512, 1.570796, 2.047618],accel_mss,speed_ms,0,blend_radius_m)
    |   speed_ms = 0.005
    |   movel([0.476821, -1.349572, -2.598463, -0.764353, 1.570796, 2.047618],accel_mss,speed_ms,0,blend_radius_m)
    |   speed_ms = 0.025
    |   movel([0.477677, -1.347959, -2.599526, -0.764904, 1.570796, 2.048473],accel_mss,speed_ms,0,blend_radius_m)
    |   movel([0.478294, -1.346339, -2.600590, -0.765460, 1.570796, 2.049091],accel_mss,speed_ms,0,blend_radius_m)
    |   movel([0.478658, -1.344752, -2.601629, -0.766008, 1.570796, 2.049454],accel_mss,speed_ms,0,blend_radius_m)
    |   movel([0.478760, -1.343233, -2.602620, -0.766537, 1.570796, 2.049556],accel_mss,speed_ms,0,blend_radius_m)
    |   movel([0.478382, -1.339736, -2.604888, -0.767764, 1.570796, 2.049178],accel_mss,speed_ms,0,blend_radius_m)
    |   movel([0.478408, -1.338690, -2.605564, -0.768135, 1.570796, 2.049205],accel_mss,speed_ms,0,blend_radius_m)
    |   movel([0.478593, -1.337680, -2.606215, -0.768494, 1.570796, 2.049389],accel_mss,speed_ms,0,blend_radius_m)
    |   movel([0.478986, -1.336760, -2.606806, -0.768823, 1.570796, 2.049782],accel_mss,speed_ms,0,blend_radius_m)
    |   movel([0.479645, -1.335982, -2.607306, -0.769101, 1.570796, 2.050441],accel_mss,speed_ms,0,blend_radius_m)
    |   movel([0.480625, -1.335334, -2.607721, -0.769334, 1.570796, 2.051421],accel_mss,speed_ms,0,blend_radius_m)
    |   movel([0.481492, -1.335098, -2.607872, -0.769419, 1.570796, 2.052289],accel_mss,speed_ms,0,blend_radius_m)
    |   movel([0.482252, -1.335197, -2.607809, -0.769383, 1.570796, 2.053048],accel_mss,speed_ms,0,blend_radius_m)
    |   movel([0.482905, -1.335552, -2.607581, -0.769256, 1.570796, 2.053701],accel_mss,speed_ms,0,blend_radius_m)
    |   movel([0.483890, -1.336704, -2.606842, -0.768843, 1.570796, 2.054687],accel_mss,speed_ms,0,blend_radius_m)
    |   movel([0.484469, -1.337923, -2.606058, -0.768408, 1.570796, 2.055265],accel_mss,speed_ms,0,blend_radius_m)
    |   movel([0.485197, -1.335855, -2.607387, -0.769147, 1.570796, 2.055994],accel_mss,speed_ms,0,blend_radius_m)
    |   movel([0.485588, -1.333878, -2.608652, -0.769859, 1.570796, 2.056384],accel_mss,speed_ms,0,blend_radius_m)
    |   movel([0.485773, -1.330063, -2.611077, -0.771248, 1.570796, 2.056569],accel_mss,speed_ms,0,blend_radius_m)
    |   movel([0.485880, -1.326195, -2.613517, -0.772677, 1.570796, 2.056677],accel_mss,speed_ms,0,blend_radius_m)
    |   movel([0.486175, -1.324147, -2.614800, -0.773442, 1.570796, 2.056971],accel_mss,speed_ms,0,blend_radius_m)
    |   movel([0.486781, -1.321976, -2.616155, -0.774258, 1.570796, 2.057577],accel_mss,speed_ms,0,blend_radius_m)
    |   movel([0.487335, -1.320582, -2.617021, -0.774786, 1.570796, 2.058131],accel_mss,speed_ms,0,blend_radius_m)
    |   movel([0.487908, -1.319452, -2.617721, -0.775216, 1.570796, 2.058704],accel_mss,speed_ms,0,blend_radius_m)
    |   movel([0.488491, -1.318572, -2.618266, -0.775552, 1.570796, 2.059287],accel_mss,speed_ms,0,blend_radius_m)
    |   movel([0.489074, -1.317931, -2.618661, -0.775797, 1.570796, 2.059870],accel_mss,speed_ms,0,blend_radius_m)
    |   movel([0.489642, -1.317515, -2.618918, -0.775956, 1.570796, 2.060439],accel_mss,speed_ms,0,blend_radius_m)
    |   movel([0.490193, -1.317306, -2.619047, -0.776037, 1.570796, 2.060989],accel_mss,speed_ms,0,blend_radius_m)
    |   movel([0.490709, -1.317289, -2.619057, -0.776043, 1.570796, 2.061506],accel_mss,speed_ms,0,blend_radius_m)
    |   movel([0.491186, -1.317453, -2.618956, -0.775980, 1.570796, 2.061982],accel_mss,speed_ms,0,blend_radius_m)
    |   movel([0.491611, -1.317781, -2.618753, -0.775854, 1.570796, 2.062408],accel_mss,speed_ms,0,blend_radius_m)
    |   movel([0.491974, -1.318257, -2.618460, -0.775672, 1.570796, 2.062770],accel_mss,speed_ms,0,blend_radius_m)
    |   movel([0.492480, -1.319590, -2.617636, -0.775163, 1.570796, 2.063276],accel_mss,speed_ms,0,blend_radius_m)
    |   movel([0.492629, -1.321327, -2.616558, -0.774504, 1.570796, 2.063426],accel_mss,speed_ms,0,blend_radius_m)
    |   movel([0.492348, -1.323346, -2.615301, -0.773742, 1.570796, 2.063144],accel_mss,speed_ms,0,blend_radius_m)
    |   movel([0.493591, -1.321653, -2.616356, -0.774380, 1.570796, 2.064387],accel_mss,speed_ms,0,blend_radius_m)
    |   movel([0.494597, -1.320010, -2.617376, -0.775003, 1.570796, 2.065393],accel_mss,speed_ms,0,blend_radius_m)
    |   movel([0.495417, -1.318404, -2.618369, -0.775616, 1.570796, 2.066213],accel_mss,speed_ms,0,blend_radius_m)
    |   movel([0.497377, -1.313599, -2.621321, -0.777469, 1.570796, 2.068173],accel_mss,speed_ms,0,blend_radius_m)
    |   movel([0.498859, -1.310219, -2.623380, -0.778791, 1.570796, 2.069655],accel_mss,speed_ms,0,blend_radius_m)
    |   movel([0.499616, -1.308827, -2.624223, -0.779339, 1.570796, 2.070412],accel_mss,speed_ms,0,blend_radius_m)
    |   movel([0.500393, -1.307640, -2.624940, -0.779809, 1.570796, 2.071190],accel_mss,speed_ms,0,blend_radius_m)
    |   movel([0.501171, -1.306658, -2.625532, -0.780199, 1.570796, 2.071967],accel_mss,speed_ms,0,blend_radius_m)
    |   movel([0.501934, -1.305878, -2.626001, -0.780510, 1.570796, 2.072731],accel_mss,speed_ms,0,blend_radius_m)
    |   movel([0.502667, -1.305294, -2.626352, -0.780743, 1.570796, 2.073464],accel_mss,speed_ms,0,blend_radius_m)
    |   movel([0.503355, -1.304905, -2.626585, -0.780899, 1.570796, 2.074152],accel_mss,speed_ms,0,blend_radius_m)
    |   movel([0.503982, -1.304707, -2.626704, -0.780978, 1.570796, 2.074779],accel_mss,speed_ms,0,blend_radius_m)
    |   movel([0.504532, -1.304696, -2.626710, -0.780982, 1.570796, 2.075329],accel_mss,speed_ms,0,blend_radius_m)
    |   movel([0.504990, -1.304870, -2.626606, -0.780913, 1.570796, 2.075786],accel_mss,speed_ms,0,blend_radius_m)
    |   movel([0.505340, -1.305221, -2.626395, -0.780772, 1.570796, 2.076136],accel_mss,speed_ms,0,blend_radius_m)
    |   movel([0.505569, -1.305747, -2.626080, -0.780562, 1.570796, 2.076366],accel_mss,speed_ms,0,blend_radius_m)
    |   movel([0.505661, -1.306444, -2.625660, -0.780284, 1.570796, 2.076458],accel_mss,speed_ms,0,blend_radius_m)
    |   movel([0.505600, -1.307307, -2.625140, -0.779941, 1.570796, 2.076396],accel_mss,speed_ms,0,blend_radius_m)
    |   movel([0.505372, -1.308332, -2.624522, -0.779535, 1.570796, 2.076168],accel_mss,speed_ms,0,blend_radius_m)
    |   movel([0.504963, -1.309512, -2.623808, -0.779069, 1.570796, 2.075759],accel_mss,speed_ms,0,blend_radius_m)
    |   movel([0.504361, -1.310843, -2.623001, -0.778545, 1.570796, 2.075158],accel_mss,speed_ms,0,blend_radius_m)
    |   movel([0.505882, -1.309678, -2.623708, -0.779003, 1.570796, 2.076678],accel_mss,speed_ms,0,blend_radius_m)
    |   movel([0.507291, -1.308414, -2.624472, -0.779502, 1.570796, 2.078088],accel_mss,speed_ms,0,blend_radius_m)
    |   movel([0.508613, -1.307071, -2.625283, -0.780035, 1.570796, 2.079409],accel_mss,speed_ms,0,blend_radius_m)
    |   movel([0.509871, -1.305667, -2.626128, -0.780594, 1.570796, 2.080667],accel_mss,speed_ms,0,blend_radius_m)
    |   movel([0.514730, -1.299885, -2.629580, -0.782925, 1.570796, 2.085526],accel_mss,speed_ms,0,blend_radius_m)
    |   movel([0.516568, -1.297775, -2.630828, -0.783786, 1.570796, 2.087364],accel_mss,speed_ms,0,blend_radius_m)
    |   movel([0.518895, -1.295391, -2.632232, -0.784766, 1.570796, 2.089692],accel_mss,speed_ms,0,blend_radius_m)
    |   movel([0.520143, -1.294383, -2.632824, -0.785183, 1.570796, 2.090940],accel_mss,speed_ms,0,blend_radius_m)
    |   movel([0.521391, -1.293655, -2.633250, -0.785484, 1.570796, 2.092187],accel_mss,speed_ms,0,blend_radius_m)
    |   movel([0.522003, -1.293434, -2.633379, -0.785576, 1.570796, 2.092800],accel_mss,speed_ms,0,blend_radius_m)
    |   movel([0.523177, -1.293343, -2.633433, -0.785614, 1.570796, 2.093973],accel_mss,speed_ms,0,blend_radius_m)
    |   movel([0.523727, -1.293507, -2.633336, -0.785546, 1.570796, 2.094523],accel_mss,speed_ms,0,blend_radius_m)
    |   movel([0.524119, -1.293909, -2.633101, -0.785379, 1.570796, 2.094915],accel_mss,speed_ms,0,blend_radius_m)
    |   movel([0.524203, -1.294537, -2.632733, -0.785119, 1.570796, 2.095000],accel_mss,speed_ms,0,blend_radius_m)
    |   movel([0.523804, -1.296075, -2.631830, -0.784484, 1.570796, 2.094600],accel_mss,speed_ms,0,blend_radius_m)
    |   movel([0.522876, -1.298205, -2.630574, -0.783610, 1.570796, 2.093672],accel_mss,speed_ms,0,blend_radius_m)
    |   movel([0.521782, -1.300323, -2.629319, -0.782746, 1.570796, 2.092578],accel_mss,speed_ms,0,blend_radius_m)
    |   movel([0.523955, -1.298870, -2.630181, -0.783338, 1.570796, 2.094752],accel_mss,speed_ms,0,blend_radius_m)
    |   movel([0.526201, -1.297582, -2.630942, -0.783865, 1.570796, 2.096997],accel_mss,speed_ms,0,blend_radius_m)
    |   movel([0.528485, -1.296466, -2.631600, -0.784323, 1.570796, 2.099281],accel_mss,speed_ms,0,blend_radius_m)
    |   movel([0.530768, -1.295526, -2.632153, -0.784710, 1.570796, 2.101564],accel_mss,speed_ms,0,blend_radius_m)
    |   movel([0.535321, -1.293655, -2.633250, -0.785484, 1.570796, 2.106117],accel_mss,speed_ms,0,blend_radius_m)
    |   movel([0.536592, -1.293226, -2.633501, -0.785662, 1.570796, 2.107388],accel_mss,speed_ms,0,blend_radius_m)
    |   movel([0.537753, -1.292944, -2.633665, -0.785779, 1.570796, 2.108550],accel_mss,speed_ms,0,blend_radius_m)
    |   movel([0.538730, -1.292873, -2.633707, -0.785809, 1.570796, 2.109526],accel_mss,speed_ms,0,blend_radius_m)
    |   movel([0.539439, -1.293071, -2.633591, -0.785727, 1.570796, 2.110235],accel_mss,speed_ms,0,blend_radius_m)
    |   movel([0.539796, -1.293629, -2.633265, -0.785495, 1.570796, 2.110592],accel_mss,speed_ms,0,blend_radius_m)
    |   movel([0.539763, -1.294477, -2.632768, -0.785143, 1.570796, 2.110560],accel_mss,speed_ms,0,blend_radius_m)
    |   movel([0.539417, -1.295518, -2.632157, -0.784713, 1.570796, 2.110214],accel_mss,speed_ms,0,blend_radius_m)
    |   movel([0.538829, -1.296650, -2.631491, -0.784247, 1.570796, 2.109626],accel_mss,speed_ms,0,blend_radius_m)
    |   movel([0.538074, -1.297775, -2.630828, -0.783786, 1.570796, 2.108870],accel_mss,speed_ms,0,blend_radius_m)
    |   movel([0.537226, -1.298794, -2.630226, -0.783369, 1.570796, 2.108023],accel_mss,speed_ms,0,blend_radius_m)
    |   movel([0.536357, -1.299608, -2.629743, -0.783037, 1.570796, 2.107154],accel_mss,speed_ms,0,blend_radius_m)
    |   movel([0.535539, -1.300121, -2.629439, -0.782829, 1.570796, 2.106335],accel_mss,speed_ms,0,blend_radius_m)
    |   movel([0.539564, -1.298618, -2.630330, -0.783441, 1.570796, 2.110360],accel_mss,speed_ms,0,blend_radius_m)
    |   movel([0.541559, -1.298052, -2.630664, -0.783672, 1.570796, 2.112356],accel_mss,speed_ms,0,blend_radius_m)
    |   movel([0.543523, -1.297629, -2.630915, -0.783846, 1.570796, 2.114320],accel_mss,speed_ms,0,blend_radius_m)
    |   movel([0.545439, -1.297358, -2.631074, -0.783957, 1.570796, 2.116236],accel_mss,speed_ms,0,blend_radius_m)
    |   movel([0.547294, -1.297255, -2.631135, -0.783999, 1.570796, 2.118090],accel_mss,speed_ms,0,blend_radius_m)
    |   movel([0.549070, -1.297333, -2.631089, -0.783967, 1.570796, 2.119867],accel_mss,speed_ms,0,blend_radius_m)
    |   movel([0.550755, -1.297601, -2.630931, -0.783857, 1.570796, 2.121552],accel_mss,speed_ms,0,blend_radius_m)
    |   movel([0.551714, -1.298079, -2.630649, -0.783661, 1.570796, 2.122511],accel_mss,speed_ms,0,blend_radius_m)
    |   movel([0.552495, -1.298983, -2.630114, -0.783292, 1.570796, 2.123291],accel_mss,speed_ms,0,blend_radius_m)
    |   movel([0.552726, -1.299550, -2.629778, -0.783061, 1.570796, 2.123522],accel_mss,speed_ms,0,blend_radius_m)
    |   movel([0.552803, -1.300169, -2.629411, -0.782809, 1.570796, 2.123599],accel_mss,speed_ms,0,blend_radius_m)
    |   movel([0.552691, -1.300824, -2.629021, -0.782543, 1.570796, 2.123487],accel_mss,speed_ms,0,blend_radius_m)
    |   movel([0.552350, -1.301497, -2.628621, -0.782270, 1.570796, 2.123146],accel_mss,speed_ms,0,blend_radius_m)
    |   movel([0.551814, -1.302079, -2.628275, -0.782035, 1.570796, 2.122610],accel_mss,speed_ms,0,blend_radius_m)
    |   movel([0.551157, -1.302554, -2.627992, -0.781844, 1.570796, 2.121954],accel_mss,speed_ms,0,blend_radius_m)
    |   movel([0.549592, -1.303332, -2.627527, -0.781530, 1.570796, 2.120389],accel_mss,speed_ms,0,blend_radius_m)
    |   movel([0.548029, -1.303757, -2.627273, -0.781359, 1.570796, 2.118825],accel_mss,speed_ms,0,blend_radius_m)
    |   movel([0.546506, -1.303910, -2.627181, -0.781298, 1.570796, 2.117302],accel_mss,speed_ms,0,blend_radius_m)
    |   movel([0.545064, -1.303868, -2.627206, -0.781315, 1.570796, 2.115860],accel_mss,speed_ms,0,blend_radius_m)
    |   movel([0.546236, -1.305031, -2.626509, -0.780848, 1.570796, 2.117032],accel_mss,speed_ms,0,blend_radius_m)
    |   movel([0.547593, -1.306014, -2.625919, -0.780456, 1.570796, 2.118389],accel_mss,speed_ms,0,blend_radius_m)
    |   movel([0.549117, -1.306810, -2.625440, -0.780139, 1.570796, 2.119913],accel_mss,speed_ms,0,blend_radius_m)
    |   movel([0.550792, -1.307414, -2.625076, -0.779899, 1.570796, 2.121588],accel_mss,speed_ms,0,blend_radius_m)
    |   movel([0.552231, -1.307696, -2.624906, -0.779787, 1.570796, 2.123027],accel_mss,speed_ms,0,blend_radius_m)
    |   movel([0.555218, -1.307960, -2.624746, -0.779682, 1.570796, 2.126015],accel_mss,speed_ms,0,blend_radius_m)
    |   movel([0.556664, -1.308230, -2.624584, -0.779575, 1.570796, 2.127460],accel_mss,speed_ms,0,blend_radius_m)
    |   movel([0.558212, -1.308690, -2.624306, -0.779393, 1.570796, 2.129009],accel_mss,speed_ms,0,blend_radius_m)
    |   movel([0.560696, -1.309649, -2.623725, -0.779015, 1.570796, 2.131492],accel_mss,speed_ms,0,blend_radius_m)
    |   movel([0.561790, -1.310255, -2.623358, -0.778776, 1.570796, 2.132586],accel_mss,speed_ms,0,blend_radius_m)
    |   movel([0.562521, -1.310911, -2.622960, -0.778519, 1.570796, 2.133318],accel_mss,speed_ms,0,blend_radius_m)
    |   movel([0.562691, -1.311249, -2.622754, -0.778386, 1.570796, 2.133487],accel_mss,speed_ms,0,blend_radius_m)
    |   movel([0.562694, -1.311591, -2.622546, -0.778252, 1.570796, 2.133490],accel_mss,speed_ms,0,blend_radius_m)
    |   movel([0.562510, -1.311931, -2.622339, -0.778119, 1.570796, 2.133307],accel_mss,speed_ms,0,blend_radius_m)
    |   movel([0.562113, -1.312265, -2.622135, -0.777989, 1.570796, 2.132910],accel_mss,speed_ms,0,blend_radius_m)
    |   movel([0.561025, -1.312830, -2.621791, -0.777768, 1.570796, 2.131822],accel_mss,speed_ms,0,blend_radius_m)
    |   movel([0.559815, -1.313224, -2.621550, -0.777614, 1.570796, 2.130611],accel_mss,speed_ms,0,blend_radius_m)
    |   movel([0.558524, -1.313482, -2.621393, -0.777514, 1.570796, 2.129320],accel_mss,speed_ms,0,blend_radius_m)
    |   movel([0.557205, -1.313629, -2.621303, -0.777457, 1.570796, 2.128001],accel_mss,speed_ms,0,blend_radius_m)
    |   movel([0.554665, -1.313702, -2.621258, -0.777429, 1.570796, 2.125461],accel_mss,speed_ms,0,blend_radius_m)
    |   movel([0.552577, -1.313666, -2.621280, -0.777443, 1.570796, 2.123374],accel_mss,speed_ms,0,blend_radius_m)
    |   movel([0.553095, -1.314568, -2.620728, -0.777093, 1.570796, 2.123892],accel_mss,speed_ms,0,blend_radius_m)
    |   movel([0.553726, -1.315378, -2.620232, -0.776779, 1.570796, 2.124522],accel_mss,speed_ms,0,blend_radius_m)
    |   movel([0.555262, -1.316761, -2.619382, -0.776246, 1.570796, 2.126058],accel_mss,speed_ms,0,blend_radius_m)
    |   movel([0.557070, -1.317890, -2.618687, -0.775813, 1.570796, 2.127867],accel_mss,speed_ms,0,blend_radius_m)
    |   movel([0.559036, -1.318840, -2.618100, -0.775449, 1.570796, 2.129832],accel_mss,speed_ms,0,blend_radius_m)
    |   movel([0.560750, -1.319486, -2.617700, -0.775203, 1.570796, 2.131546],accel_mss,speed_ms,0,blend_radius_m)
    |   movel([0.566077, -1.321158, -2.616663, -0.774568, 1.570796, 2.136873],accel_mss,speed_ms,0,blend_radius_m)
    |   movel([0.566925, -1.321690, -2.616333, -0.774366, 1.570796, 2.137721],accel_mss,speed_ms,0,blend_radius_m)
    |   movel([0.567404, -1.322414, -2.615882, -0.774093, 1.570796, 2.138201],accel_mss,speed_ms,0,blend_radius_m)
    |   movel([0.567376, -1.322780, -2.615654, -0.773955, 1.570796, 2.138172],accel_mss,speed_ms,0,blend_radius_m)
    |   movel([0.567099, -1.323110, -2.615448, -0.773831, 1.570796, 2.137895],accel_mss,speed_ms,0,blend_radius_m)
    |   movel([0.566520, -1.323378, -2.615281, -0.773730, 1.570796, 2.137317],accel_mss,speed_ms,0,blend_radius_m)
    |   movel([0.565588, -1.323554, -2.615171, -0.773664, 1.570796, 2.136384],accel_mss,speed_ms,0,blend_radius_m)
    |   movel([0.564160, -1.323615, -2.615133, -0.773641, 1.570796, 2.134956],accel_mss,speed_ms,0,blend_radius_m)
    |   movel([0.562620, -1.323495, -2.615208, -0.773686, 1.570796, 2.133416],accel_mss,speed_ms,0,blend_radius_m)
    |   movel([0.561231, -1.323153, -2.615421, -0.773815, 1.570796, 2.132027],accel_mss,speed_ms,0,blend_radius_m)
    |   movel([0.560674, -1.322887, -2.615587, -0.773915, 1.570796, 2.131470],accel_mss,speed_ms,0,blend_radius_m)
    |   movel([0.560257, -1.322548, -2.615798, -0.774042, 1.570796, 2.131053],accel_mss,speed_ms,0,blend_radius_m)
    |   movel([0.561241, -1.324942, -2.614303, -0.773144, 1.570796, 2.132038],accel_mss,speed_ms,0,blend_radius_m)
    |   movel([0.562524, -1.327120, -2.612935, -0.772333, 1.570796, 2.133321],accel_mss,speed_ms,0,blend_radius_m)
    |   movel([0.564045, -1.329119, -2.611675, -0.771595, 1.570796, 2.134841],accel_mss,speed_ms,0,blend_radius_m)
    |   movel([0.565745, -1.330982, -2.610496, -0.770912, 1.570796, 2.136541],accel_mss,speed_ms,0,blend_radius_m)
    |   movel([0.569451, -1.334431, -2.608299, -0.769659, 1.570796, 2.140247],accel_mss,speed_ms,0,blend_radius_m)
    |   movel([0.573175, -1.337754, -2.606167, -0.768468, 1.570796, 2.143972],accel_mss,speed_ms,0,blend_radius_m)
    |   movel([0.573691, -1.338478, -2.605701, -0.768210, 1.570796, 2.144487],accel_mss,speed_ms,0,blend_radius_m)
    |   movel([0.573735, -1.338932, -2.605408, -0.768049, 1.570796, 2.144531],accel_mss,speed_ms,0,blend_radius_m)
    |   movel([0.573528, -1.339439, -2.605080, -0.767869, 1.570796, 2.144324],accel_mss,speed_ms,0,blend_radius_m)
    |   movel([0.573099, -1.339888, -2.604790, -0.767711, 1.570796, 2.143896],accel_mss,speed_ms,0,blend_radius_m)
    |   movel([0.571722, -1.340678, -2.604279, -0.767432, 1.570796, 2.142518],accel_mss,speed_ms,0,blend_radius_m)
    |   movel([0.570874, -1.341000, -2.604070, -0.767318, 1.570796, 2.141670],accel_mss,speed_ms,0,blend_radius_m)
    |   movel([0.569183, -1.341339, -2.603851, -0.767199, 1.570796, 2.139979],accel_mss,speed_ms,0,blend_radius_m)
    |   movel([0.567539, -1.341325, -2.603860, -0.767204, 1.570796, 2.138335],accel_mss,speed_ms,0,blend_radius_m)
    |   movel([0.565973, -1.341026, -2.604053, -0.767309, 1.570796, 2.136769],accel_mss,speed_ms,0,blend_radius_m)
    |   movel([0.564526, -1.340506, -2.604390, -0.767492, 1.570796, 2.135323],accel_mss,speed_ms,0,blend_radius_m)
    |   movel([0.563234, -1.339833, -2.604826, -0.767730, 1.570796, 2.134030],accel_mss,speed_ms,0,blend_radius_m)
    |   movel([0.562135, -1.339068, -2.605320, -0.768001, 1.570796, 2.132931],accel_mss,speed_ms,0,blend_radius_m)
    |   movel([0.561270, -1.338276, -2.605831, -0.768282, 1.570796, 2.132067],accel_mss,speed_ms,0,blend_radius_m)
    |   movel([0.561003, -1.338714, -2.605548, -0.768126, 1.570796, 2.131799],accel_mss,speed_ms,0,blend_radius_m)
    |   movel([0.560974, -1.339164, -2.605258, -0.767967, 1.570796, 2.131770],accel_mss,speed_ms,0,blend_radius_m)
    |   movel([0.561152, -1.340097, -2.604655, -0.767637, 1.570796, 2.131948],accel_mss,speed_ms,0,blend_radius_m)
    |   movel([0.561472, -1.340950, -2.604103, -0.767336, 1.570796, 2.132269],accel_mss,speed_ms,0,blend_radius_m)
    |   movel([0.562363, -1.342502, -2.603095, -0.766792, 1.570796, 2.133160],accel_mss,speed_ms,0,blend_radius_m)
    |   movel([0.564091, -1.345024, -2.601451, -0.765914, 1.570796, 2.134887],accel_mss,speed_ms,0,blend_radius_m)
    |   movel([0.565937, -1.347426, -2.599877, -0.765086, 1.570796, 2.136734],accel_mss,speed_ms,0,blend_radius_m)
    |   movel([0.569942, -1.351936, -2.596899, -0.763554, 1.570796, 2.140738],accel_mss,speed_ms,0,blend_radius_m)
    |   movel([0.571032, -1.353216, -2.596049, -0.763124, 1.570796, 2.141829],accel_mss,speed_ms,0,blend_radius_m)
    |   movel([0.571656, -1.354143, -2.595432, -0.762814, 1.570796, 2.142452],accel_mss,speed_ms,0,blend_radius_m)
    |   movel([0.572170, -1.355176, -2.594743, -0.762470, 1.570796, 2.142967],accel_mss,speed_ms,0,blend_radius_m)
    |   movel([0.572449, -1.356251, -2.594024, -0.762114, 1.570796, 2.143245],accel_mss,speed_ms,0,blend_radius_m)
    |   movel([0.572374, -1.357299, -2.593321, -0.761768, 1.570796, 2.143170],accel_mss,speed_ms,0,blend_radius_m)
    |   movel([0.572168, -1.357794, -2.592990, -0.761606, 1.570796, 2.142964],accel_mss,speed_ms,0,blend_radius_m)
    |   movel([0.571829, -1.358259, -2.592677, -0.761453, 1.570796, 2.142626],accel_mss,speed_ms,0,blend_radius_m)
    |   movel([0.571338, -1.358686, -2.592390, -0.761313, 1.570796, 2.142135],accel_mss,speed_ms,0,blend_radius_m)
    |   movel([0.570686, -1.359068, -2.592133, -0.761188, 1.570796, 2.141483],accel_mss,speed_ms,0,blend_radius_m)
    |   movel([0.569974, -1.359179, -2.592058, -0.761152, 1.570796, 2.140771],accel_mss,speed_ms,0,blend_radius_m)
    |   movel([0.569174, -1.359018, -2.592167, -0.761205, 1.570796, 2.139971],accel_mss,speed_ms,0,blend_radius_m)
    |   movel([0.565202, -1.357551, -2.593152, -0.761685, 1.570796, 2.135998],accel_mss,speed_ms,0,blend_radius_m)
    |   movel([0.563995, -1.356820, -2.593642, -0.761926, 1.570796, 2.134792],accel_mss,speed_ms,0,blend_radius_m)
    |   movel([0.563549, -1.356378, -2.593939, -0.762072, 1.570796, 2.134345],accel_mss,speed_ms,0,blend_radius_m)
    |   movel([0.563259, -1.355871, -2.594278, -0.762240, 1.570796, 2.134055],accel_mss,speed_ms,0,blend_radius_m)
    |   movel([0.563894, -1.359000, -2.592178, -0.761210, 1.570796, 2.134690],accel_mss,speed_ms,0,blend_radius_m)
    |   movel([0.564930, -1.361895, -2.590224, -0.760271, 1.570796, 2.135727],accel_mss,speed_ms,0,blend_radius_m)
    |   movel([0.566288, -1.364581, -2.588399, -0.759409, 1.570796, 2.137084],accel_mss,speed_ms,0,blend_radius_m)
    |   movel([0.567890, -1.367082, -2.586691, -0.758616, 1.570796, 2.138687],accel_mss,speed_ms,0,blend_radius_m)
    |   movel([0.569508, -1.368812, -2.585505, -0.758073, 1.570796, 2.140304],accel_mss,speed_ms,0,blend_radius_m)
    |   movel([0.571786, -1.371355, -2.583753, -0.757281, 1.570796, 2.142582],accel_mss,speed_ms,0,blend_radius_m)
    |   movel([0.572698, -1.372726, -2.582804, -0.756859, 1.570796, 2.143494],accel_mss,speed_ms,0,blend_radius_m)
    |   movel([0.573213, -1.374054, -2.581883, -0.756452, 1.570796, 2.144009],accel_mss,speed_ms,0,blend_radius_m)
    |   movel([0.573263, -1.374675, -2.581452, -0.756263, 1.570796, 2.144060],accel_mss,speed_ms,0,blend_radius_m)
    |   movel([0.573144, -1.375252, -2.581050, -0.756087, 1.570796, 2.143941],accel_mss,speed_ms,0,blend_radius_m)
    |   movel([0.572832, -1.375778, -2.580683, -0.755928, 1.570796, 2.143628],accel_mss,speed_ms,0,blend_radius_m)
    |   movel([0.572309, -1.376242, -2.580360, -0.755787, 1.570796, 2.143105],accel_mss,speed_ms,0,blend_radius_m)
    |   movel([0.571702, -1.376584, -2.580121, -0.755684, 1.570796, 2.142498],accel_mss,speed_ms,0,blend_radius_m)
    |   movel([0.571079, -1.376828, -2.579951, -0.755610, 1.570796, 2.141875],accel_mss,speed_ms,0,blend_radius_m)
    |   movel([0.569831, -1.377119, -2.579747, -0.755523, 1.570796, 2.140627],accel_mss,speed_ms,0,blend_radius_m)
    |   movel([0.568531, -1.377283, -2.579632, -0.755473, 1.570796, 2.139327],accel_mss,speed_ms,0,blend_radius_m)
    |   movel([0.566060, -1.377286, -2.579631, -0.755473, 1.570796, 2.136857],accel_mss,speed_ms,0,blend_radius_m)
    |   movel([0.564904, -1.377127, -2.579742, -0.755520, 1.570796, 2.135700],accel_mss,speed_ms,0,blend_radius_m)
    |   movel([0.566200, -1.378941, -2.578471, -0.754977, 1.570796, 2.136997],accel_mss,speed_ms,0,blend_radius_m)
    |   movel([0.567641, -1.380619, -2.577292, -0.754478, 1.570796, 2.138437],accel_mss,speed_ms,0,blend_radius_m)
    |   movel([0.569208, -1.382177, -2.576193, -0.754019, 1.570796, 2.140004],accel_mss,speed_ms,0,blend_radius_m)
    |   movel([0.570887, -1.383627, -2.575167, -0.753594, 1.570796, 2.141683],accel_mss,speed_ms,0,blend_radius_m)
    |   movel([0.574515, -1.386268, -2.573291, -0.752829, 1.570796, 2.145311],accel_mss,speed_ms,0,blend_radius_m)
    |   movel([0.578407, -1.388652, -2.571589, -0.752148, 1.570796, 2.149203],accel_mss,speed_ms,0,blend_radius_m)
    |   movel([0.579346, -1.389428, -2.571034, -0.751928, 1.570796, 2.150143],accel_mss,speed_ms,0,blend_radius_m)
    |   movel([0.579550, -1.389960, -2.570652, -0.751777, 1.570796, 2.150347],accel_mss,speed_ms,0,blend_radius_m)
    |   movel([0.579414, -1.390611, -2.570185, -0.751594, 1.570796, 2.150210],accel_mss,speed_ms,0,blend_radius_m)
    |   movel([0.579137, -1.391041, -2.569875, -0.751473, 1.570796, 2.149933],accel_mss,speed_ms,0,blend_radius_m)
    |   movel([0.578763, -1.391416, -2.569605, -0.751367, 1.570796, 2.149560],accel_mss,speed_ms,0,blend_radius_m)
    |   movel([0.577769, -1.392026, -2.569166, -0.751197, 1.570796, 2.148566],accel_mss,speed_ms,0,blend_radius_m)
    |   movel([0.576546, -1.392460, -2.568853, -0.751076, 1.570796, 2.147343],accel_mss,speed_ms,0,blend_radius_m)
    |   movel([0.575200, -1.392746, -2.568647, -0.750996, 1.570796, 2.145996],accel_mss,speed_ms,0,blend_radius_m)
    |   movel([0.572584, -1.392961, -2.568492, -0.750936, 1.570796, 2.143381],accel_mss,speed_ms,0,blend_radius_m)
    |   movel([0.570809, -1.392845, -2.568576, -0.750969, 1.570796, 2.141605],accel_mss,speed_ms,0,blend_radius_m)
    |   movel([0.571535, -1.393443, -2.568143, -0.750802, 1.570796, 2.142331],accel_mss,speed_ms,0,blend_radius_m)
    |   movel([0.572349, -1.393945, -2.567780, -0.750663, 1.570796, 2.143145],accel_mss,speed_ms,0,blend_radius_m)
    |   movel([0.574202, -1.394682, -2.567247, -0.750460, 1.570796, 2.144998],accel_mss,speed_ms,0,blend_radius_m)
    |   movel([0.576313, -1.395072, -2.566965, -0.750353, 1.570796, 2.147110],accel_mss,speed_ms,0,blend_radius_m)
    |   movel([0.578620, -1.395143, -2.566913, -0.750333, 1.570796, 2.149417],accel_mss,speed_ms,0,blend_radius_m)
    |   movel([0.581071, -1.394908, -2.567083, -0.750398, 1.570796, 2.151867],accel_mss,speed_ms,0,blend_radius_m)
    |   movel([0.583605, -1.394395, -2.567455, -0.750539, 1.570796, 2.154401],accel_mss,speed_ms,0,blend_radius_m)
    |   movel([0.586169, -1.393616, -2.568018, -0.750754, 1.570796, 2.156965],accel_mss,speed_ms,0,blend_radius_m)
    |   movel([0.588706, -1.392596, -2.568755, -0.751038, 1.570796, 2.159502],accel_mss,speed_ms,0,blend_radius_m)
    |   movel([0.589829, -1.392133, -2.569089, -0.751167, 1.570796, 2.160625],accel_mss,speed_ms,0,blend_radius_m)
    |   movel([0.590366, -1.392015, -2.569174, -0.751200, 1.570796, 2.161163],accel_mss,speed_ms,0,blend_radius_m)
    |   movel([0.590849, -1.392039, -2.569157, -0.751193, 1.570796, 2.161645],accel_mss,speed_ms,0,blend_radius_m)
    |   movel([0.591241, -1.392269, -2.568991, -0.751129, 1.570796, 2.162037],accel_mss,speed_ms,0,blend_radius_m)
    |   movel([0.591481, -1.392641, -2.568723, -0.751025, 1.570796, 2.162277],accel_mss,speed_ms,0,blend_radius_m)
    |   movel([0.591567, -1.393380, -2.568189, -0.750820, 1.570796, 2.162364],accel_mss,speed_ms,0,blend_radius_m)
    |   movel([0.591345, -1.394278, -2.567539, -0.750571, 1.570796, 2.162141],accel_mss,speed_ms,0,blend_radius_m)
    |   movel([0.590881, -1.395278, -2.566815, -0.750296, 1.570796, 2.161677],accel_mss,speed_ms,0,blend_radius_m)
    |   movel([0.590241, -1.396332, -2.566049, -0.750007, 1.570796, 2.161037],accel_mss,speed_ms,0,blend_radius_m)
    |   movel([0.588704, -1.398382, -2.564556, -0.749451, 1.570796, 2.159500],accel_mss,speed_ms,0,blend_radius_m)
    |   movel([0.587266, -1.400014, -2.563363, -0.749012, 1.570796, 2.158063],accel_mss,speed_ms,0,blend_radius_m)
    |   movel([0.589604, -1.398798, -2.564252, -0.749339, 1.570796, 2.160401],accel_mss,speed_ms,0,blend_radius_m)
    |   movel([0.591861, -1.397382, -2.565285, -0.749722, 1.570796, 2.162657],accel_mss,speed_ms,0,blend_radius_m)
    |   movel([0.594018, -1.395784, -2.566448, -0.750157, 1.570796, 2.164815],accel_mss,speed_ms,0,blend_radius_m)
    |   movel([0.596054, -1.394033, -2.567717, -0.750639, 1.570796, 2.166851],accel_mss,speed_ms,0,blend_radius_m)
    |   movel([0.597944, -1.392152, -2.569076, -0.751162, 1.570796, 2.168740],accel_mss,speed_ms,0,blend_radius_m)
    |   movel([0.599672, -1.390163, -2.570506, -0.751720, 1.570796, 2.170468],accel_mss,speed_ms,0,blend_radius_m)
    |   movel([0.601208, -1.388096, -2.571987, -0.752306, 1.570796, 2.172005],accel_mss,speed_ms,0,blend_radius_m)
    |   movel([0.602535, -1.385972, -2.573502, -0.752915, 1.570796, 2.173331],accel_mss,speed_ms,0,blend_radius_m)
    |   movel([0.604026, -1.382955, -2.575643, -0.753791, 1.570796, 2.174823],accel_mss,speed_ms,0,blend_radius_m)
    |   movel([0.604912, -1.381390, -2.576749, -0.754250, 1.570796, 2.175709],accel_mss,speed_ms,0,blend_radius_m)
    |   movel([0.605419, -1.380685, -2.577246, -0.754459, 1.570796, 2.176215],accel_mss,speed_ms,0,blend_radius_m)
    |   movel([0.605977, -1.380066, -2.577681, -0.754642, 1.570796, 2.176773],accel_mss,speed_ms,0,blend_radius_m)
    |   movel([0.606991, -1.379225, -2.578272, -0.754892, 1.570796, 2.177787],accel_mss,speed_ms,0,blend_radius_m)
    |   movel([0.607714, -1.378895, -2.578504, -0.754991, 1.570796, 2.178510],accel_mss,speed_ms,0,blend_radius_m)
    |   movel([0.608206, -1.378963, -2.578456, -0.754970, 1.570796, 2.179003],accel_mss,speed_ms,0,blend_radius_m)
    |   movel([0.608528, -1.379314, -2.578209, -0.754866, 1.570796, 2.179324],accel_mss,speed_ms,0,blend_radius_m)
    |   movel([0.609045, -1.380931, -2.577072, -0.754386, 1.570796, 2.179841],accel_mss,speed_ms,0,blend_radius_m)
    |   movel([0.609266, -1.381278, -2.576827, -0.754283, 1.570796, 2.180062],accel_mss,speed_ms,0,blend_radius_m)
    |   movel([0.610734, -1.380000, -2.577727, -0.754662, 1.570796, 2.181531],accel_mss,speed_ms,0,blend_radius_m)
    |   movel([0.612120, -1.378620, -2.578696, -0.755073, 1.570796, 2.182916],accel_mss,speed_ms,0,blend_radius_m)
    |   movel([0.613422, -1.377152, -2.579724, -0.755513, 1.570796, 2.184219],accel_mss,speed_ms,0,blend_radius_m)
    |   movel([0.614645, -1.375605, -2.580804, -0.755980, 1.570796, 2.185441],accel_mss,speed_ms,0,blend_radius_m)
    |   movel([0.615782, -1.373995, -2.581924, -0.756470, 1.570796, 2.186578],accel_mss,speed_ms,0,blend_radius_m)
    |   movel([0.616837, -1.372330, -2.583079, -0.756981, 1.570796, 2.187633],accel_mss,speed_ms,0,blend_radius_m)
    |   movel([0.618706, -1.368889, -2.585451, -0.758048, 1.570796, 2.189502],accel_mss,speed_ms,0,blend_radius_m)
    |   movel([0.620245, -1.365388, -2.587849, -0.759152, 1.570796, 2.191041],accel_mss,speed_ms,0,blend_radius_m)
    |   movel([0.621460, -1.361927, -2.590202, -0.760260, 1.570796, 2.192256],accel_mss,speed_ms,0,blend_radius_m)
    |   movel([0.622342, -1.358612, -2.592439, -0.761337, 1.570796, 2.193139],accel_mss,speed_ms,0,blend_radius_m)
    |   movel([0.622897, -1.355551, -2.594492, -0.762346, 1.570796, 2.193694],accel_mss,speed_ms,0,blend_radius_m)
    |   speed_ms = 0.005
    |   movel([0.622897, -1.346560, -2.590392, -0.775437, 1.570796, 2.193694],accel_mss,speed_ms,0,blend_radius_m)
    |   speed_ms = 0.040
    |   movel([0.610502, -1.345377, -2.591171, -0.775841, 1.570796, 2.181298],accel_mss,speed_ms,0,blend_radius_m)
    |   speed_ms = 0.005
    |   movel([0.610502, -1.354376, -2.595276, -0.762737, 1.570796, 2.181298],accel_mss,speed_ms,0,blend_radius_m)
    |   speed_ms = 0.025
    |   movel([0.610066, -1.353065, -2.596149, -0.763175, 1.570796, 2.180862],accel_mss,speed_ms,0,blend_radius_m)
    |   movel([0.609319, -1.351998, -2.596858, -0.763533, 1.570796, 2.180115],accel_mss,speed_ms,0,blend_radius_m)
    |   movel([0.608310, -1.351150, -2.597420, -0.763819, 1.570796, 2.179106],accel_mss,speed_ms,0,blend_radius_m)
    |   movel([0.607093, -1.350494, -2.597854, -0.764041, 1.570796, 2.177889],accel_mss,speed_ms,0,blend_radius_m)
    |   movel([0.605719, -1.350002, -2.598179, -0.764207, 1.570796, 2.176515],accel_mss,speed_ms,0,blend_radius_m)
    |   movel([0.604238, -1.349647, -2.598414, -0.764328, 1.570796, 2.175034],accel_mss,speed_ms,0,blend_radius_m)
    |   movel([0.601170, -1.349236, -2.598685, -0.764468, 1.570796, 2.171966],accel_mss,speed_ms,0,blend_radius_m)
    |   speed_ms = 0.005
    |   movel([0.601170, -1.340202, -2.594557, -0.777630, 1.570796, 2.171966],accel_mss,speed_ms,0,blend_radius_m)
    |   speed_ms = 0.040
    |   movel([0.605361, -1.340299, -2.594494, -0.777596, 1.570796, 2.176157],accel_mss,speed_ms,0,blend_radius_m)
    |   speed_ms = 0.005
    |   movel([0.605361, -1.349332, -2.598622, -0.764435, 1.570796, 2.176157],accel_mss,speed_ms,0,blend_radius_m)
    |   speed_ms = 0.025
    |   movel([0.606903, -1.347649, -2.599730, -0.765010, 1.570796, 2.177699],accel_mss,speed_ms,0,blend_radius_m)
    |   movel([0.608271, -1.345949, -2.600846, -0.765595, 1.570796, 2.179067],accel_mss,speed_ms,0,blend_radius_m)
    |   movel([0.609470, -1.344228, -2.601971, -0.766190, 1.570796, 2.180267],accel_mss,speed_ms,0,blend_radius_m)
    |   movel([0.610511, -1.342486, -2.603105, -0.766797, 1.570796, 2.181308],accel_mss,speed_ms,0,blend_radius_m)
    |   movel([0.611405, -1.340723, -2.604250, -0.767416, 1.570796, 2.182201],accel_mss,speed_ms,0,blend_radius_m)
    |   movel([0.612159, -1.338937, -2.605405, -0.768047, 1.570796, 2.182955],accel_mss,speed_ms,0,blend_radius_m)
    |   movel([0.612782, -1.337127, -2.606570, -0.768691, 1.570796, 2.183579],accel_mss,speed_ms,0,blend_radius_m)
    |   movel([0.613285, -1.335293, -2.607747, -0.769349, 1.570796, 2.184082],accel_mss,speed_ms,0,blend_radius_m)
    |   movel([0.614347, -1.329963, -2.611141, -0.771285, 1.570796, 2.185143],accel_mss,speed_ms,0,blend_radius_m)
    |   movel([0.614957, -1.327383, -2.612770, -0.772236, 1.570796, 2.185753],accel_mss,speed_ms,0,blend_radius_m)
    |   movel([0.615950, -1.324518, -2.614568, -0.773302, 1.570796, 2.186746],accel_mss,speed_ms,0,blend_radius_m)
    |   movel([0.617539, -1.320905, -2.616820, -0.774663, 1.570796, 2.188336],accel_mss,speed_ms,0,blend_radius_m)
    |   movel([0.619412, -1.317279, -2.619063, -0.776047, 1.570796, 2.190208],accel_mss,speed_ms,0,blend_radius_m)
    |   movel([0.621631, -1.313688, -2.621267, -0.777434, 1.570796, 2.192427],accel_mss,speed_ms,0,blend_radius_m)
    |   movel([0.622890, -1.311921, -2.622345, -0.778123, 1.570796, 2.193686],accel_mss,speed_ms,0,blend_radius_m)
    |   movel([0.624259, -1.310184, -2.623400, -0.778804, 1.570796, 2.195056],accel_mss,speed_ms,0,blend_radius_m)
    |   movel([0.626580, -1.307633, -2.624944, -0.779812, 1.570796, 2.197376],accel_mss,speed_ms,0,blend_radius_m)
    |   movel([0.629067, -1.305352, -2.626317, -0.780720, 1.570796, 2.199863],accel_mss,speed_ms,0,blend_radius_m)
    |   movel([0.631695, -1.303353, -2.627514, -0.781522, 1.570796, 2.202491],accel_mss,speed_ms,0,blend_radius_m)
    |   movel([0.634436, -1.301648, -2.628531, -0.782209, 1.570796, 2.205232],accel_mss,speed_ms,0,blend_radius_m)
    |   movel([0.637256, -1.300253, -2.629361, -0.782775, 1.570796, 2.208052],accel_mss,speed_ms,0,blend_radius_m)
    |   movel([0.640128, -1.299181, -2.629997, -0.783211, 1.570796, 2.210925],accel_mss,speed_ms,0,blend_radius_m)
    |   movel([0.643026, -1.298442, -2.630434, -0.783513, 1.570796, 2.213822],accel_mss,speed_ms,0,blend_radius_m)
    |   movel([0.645914, -1.298048, -2.630667, -0.783674, 1.570796, 2.216711],accel_mss,speed_ms,0,blend_radius_m)
    |   movel([0.648024, -1.297993, -2.630700, -0.783697, 1.570796, 2.218820],accel_mss,speed_ms,0,blend_radius_m)
    |   movel([0.650051, -1.298145, -2.630609, -0.783634, 1.570796, 2.220848],accel_mss,speed_ms,0,blend_radius_m)
    |   movel([0.651979, -1.298499, -2.630400, -0.783490, 1.570796, 2.222776],accel_mss,speed_ms,0,blend_radius_m)
    |   movel([0.653801, -1.299040, -2.630080, -0.783269, 1.570796, 2.224597],accel_mss,speed_ms,0,blend_radius_m)
    |   movel([0.655496, -1.299767, -2.629649, -0.782973, 1.570796, 2.226292],accel_mss,speed_ms,0,blend_radius_m)
    |   movel([0.657053, -1.300666, -2.629116, -0.782607, 1.570796, 2.227849],accel_mss,speed_ms,0,blend_radius_m)
    |   movel([0.658458, -1.301728, -2.628484, -0.782177, 1.570796, 2.229254],accel_mss,speed_ms,0,blend_radius_m)
    |   movel([0.659698, -1.302944, -2.627759, -0.781686, 1.570796, 2.230494],accel_mss,speed_ms,0,blend_radius_m)
    |   movel([0.660758, -1.304304, -2.626945, -0.781140, 1.570796, 2.231554],accel_mss,speed_ms,0,blend_radius_m)
    |   movel([0.661630, -1.305798, -2.626049, -0.780542, 1.570796, 2.232426],accel_mss,speed_ms,0,blend_radius_m)
    |   movel([0.662298, -1.307417, -2.625075, -0.779898, 1.570796, 2.233095],accel_mss,speed_ms,0,blend_radius_m)
    |   movel([0.662753, -1.309151, -2.624027, -0.779211, 1.570796, 2.233549],accel_mss,speed_ms,0,blend_radius_m)
    |   movel([0.662982, -1.310989, -2.622912, -0.778488, 1.570796, 2.233779],accel_mss,speed_ms,0,blend_radius_m)
    |   movel([0.662971, -1.312923, -2.621734, -0.777732, 1.570796, 2.233767],accel_mss,speed_ms,0,blend_radius_m)
    |   movel([0.662713, -1.314939, -2.620501, -0.776949, 1.570796, 2.233509],accel_mss,speed_ms,0,blend_radius_m)
    |   movel([0.662194, -1.317034, -2.619214, -0.776141, 1.570796, 2.232990],accel_mss,speed_ms,0,blend_radius_m)
    |   movel([0.661222, -1.319798, -2.617507, -0.775084, 1.570796, 2.232018],accel_mss,speed_ms,0,blend_radius_m)
    |   movel([0.660038, -1.322566, -2.615787, -0.774036, 1.570796, 2.230834],accel_mss,speed_ms,0,blend_radius_m)
    |   movel([0.658688, -1.325329, -2.614061, -0.773000, 1.570796, 2.229485],accel_mss,speed_ms,0,blend_radius_m)
    |   movel([0.657229, -1.328072, -2.612336, -0.771981, 1.570796, 2.228025],accel_mss,speed_ms,0,blend_radius_m)
    |   movel([0.653850, -1.333959, -2.608600, -0.769830, 1.570796, 2.224647],accel_mss,speed_ms,0,blend_radius_m)
    |   movel([0.650268, -1.339770, -2.604866, -0.767752, 1.570796, 2.221064],accel_mss,speed_ms,0,blend_radius_m)
    |   movel([0.646532, -1.345512, -2.601132, -0.765745, 1.570796, 2.217329],accel_mss,speed_ms,0,blend_radius_m)
    |   movel([0.642701, -1.351180, -2.597400, -0.763809, 1.570796, 2.213498],accel_mss,speed_ms,0,blend_radius_m)
    |   movel([0.627487, -1.373203, -2.582474, -0.756712, 1.570796, 2.198284],accel_mss,speed_ms,0,blend_radius_m)
    |   movel([0.620438, -1.383934, -2.574950, -0.753505, 1.570796, 2.191235],accel_mss,speed_ms,0,blend_radius_m)
    |   movel([0.617107, -1.389270, -2.571147, -0.751972, 1.570796, 2.187903],accel_mss,speed_ms,0,blend_radius_m)
    |   movel([0.613962, -1.394580, -2.567321, -0.750488, 1.570796, 2.184759],accel_mss,speed_ms,0,blend_radius_m)
    |   movel([0.611040, -1.399864, -2.563473, -0.749052, 1.570796, 2.181837],accel_mss,speed_ms,0,blend_radius_m)
    |   movel([0.608382, -1.405119, -2.559605, -0.747665, 1.570796, 2.179179],accel_mss,speed_ms,0,blend_radius_m)
    |   movel([0.606022, -1.410342, -2.555720, -0.746327, 1.570796, 2.176819],accel_mss,speed_ms,0,blend_radius_m)
    |   movel([0.604002, -1.415533, -2.551818, -0.745037, 1.570796, 2.174798],accel_mss,speed_ms,0,blend_radius_m)
    |   movel([0.603351, -1.417541, -2.550299, -0.744549, 1.570796, 2.174148],accel_mss,speed_ms,0,blend_radius_m)
    |   movel([0.602934, -1.419507, -2.548805, -0.744078, 1.570796, 2.173730],accel_mss,speed_ms,0,blend_radius_m)
    |   movel([0.602913, -1.421316, -2.547425, -0.743648, 1.570796, 2.173709],accel_mss,speed_ms,0,blend_radius_m)
    |   movel([0.603103, -1.422127, -2.546805, -0.743457, 1.570796, 2.173899],accel_mss,speed_ms,0,blend_radius_m)
    |   movel([0.603457, -1.422856, -2.546246, -0.743287, 1.570796, 2.174253],accel_mss,speed_ms,0,blend_radius_m)
    |   speed_ms = 0.005
    |   movel([0.603457, -1.414356, -2.542440, -0.755592, 1.570796, 2.174253],accel_mss,speed_ms,0,blend_radius_m)
    |   speed_ms = 0.040
    |   movel([0.603863, -1.383508, -2.565076, -0.763806, 1.570796, 2.174659],accel_mss,speed_ms,0,blend_radius_m)
    |   speed_ms = 0.005
    |   movel([0.603863, -1.392238, -2.569014, -0.751138, 1.570796, 2.174659],accel_mss,speed_ms,0,blend_radius_m)
    |   speed_ms = 0.025
    |   movel([0.603127, -1.392685, -2.568691, -0.751013, 1.570796, 2.173924],accel_mss,speed_ms,0,blend_radius_m)
    |   movel([0.602452, -1.393269, -2.568270, -0.750851, 1.570796, 2.173248],accel_mss,speed_ms,0,blend_radius_m)
    |   movel([0.601838, -1.393967, -2.567765, -0.750657, 1.570796, 2.172634],accel_mss,speed_ms,0,blend_radius_m)
    |   movel([0.601271, -1.394766, -2.567186, -0.750437, 1.570796, 2.172067],accel_mss,speed_ms,0,blend_radius_m)
    |   movel([0.600275, -1.396590, -2.565862, -0.749937, 1.570796, 2.171071],accel_mss,speed_ms,0,blend_radius_m)
    |   movel([0.599419, -1.398598, -2.564398, -0.749393, 1.570796, 2.170215],accel_mss,speed_ms,0,blend_radius_m)
    |   movel([0.597252, -1.404343, -2.560179, -0.747867, 1.570796, 2.168049],accel_mss,speed_ms,0,blend_radius_m)
    |   movel([0.596512, -1.405711, -2.559167, -0.747512, 1.570796, 2.167309],accel_mss,speed_ms,0,blend_radius_m)
    |   movel([0.596041, -1.406232, -2.558780, -0.747377, 1.570796, 2.166837],accel_mss,speed_ms,0,blend_radius_m)
    |   movel([0.595523, -1.406503, -2.558579, -0.747307, 1.570796, 2.166319],accel_mss,speed_ms,0,blend_radius_m)
    |   movel([0.595134, -1.406544, -2.558549, -0.747296, 1.570796, 2.165930],accel_mss,speed_ms,0,blend_radius_m)
    |   movel([0.594860, -1.406384, -2.558668, -0.747337, 1.570796, 2.165656],accel_mss,speed_ms,0,blend_radius_m)
    |   movel([0.594686, -1.406051, -2.558915, -0.747423, 1.570796, 2.165483],accel_mss,speed_ms,0,blend_radius_m)
    |   movel([0.594599, -1.404973, -2.559712, -0.747703, 1.570796, 2.165395],accel_mss,speed_ms,0,blend_radius_m)
    |   movel([0.594773, -1.403540, -2.560772, -0.748078, 1.570796, 2.165569],accel_mss,speed_ms,0,blend_radius_m)
    |   movel([0.595504, -1.400500, -2.563007, -0.748882, 1.570796, 2.166300],accel_mss,speed_ms,0,blend_radius_m)
    |   movel([0.596090, -1.398758, -2.564281, -0.749349, 1.570796, 2.166886],accel_mss,speed_ms,0,blend_radius_m)
    |   movel([0.594372, -1.400820, -2.562772, -0.748797, 1.570796, 2.165169],accel_mss,speed_ms,0,blend_radius_m)
    |   movel([0.592915, -1.402977, -2.561186, -0.748226, 1.570796, 2.163712],accel_mss,speed_ms,0,blend_radius_m)
    |   movel([0.591689, -1.405202, -2.559544, -0.747644, 1.570796, 2.162485],accel_mss,speed_ms,0,blend_radius_m)
    |   movel([0.590673, -1.407457, -2.557871, -0.747061, 1.570796, 2.161469],accel_mss,speed_ms,0,blend_radius_m)
    |   movel([0.589835, -1.409717, -2.556187, -0.746485, 1.570796, 2.160631],accel_mss,speed_ms,0,blend_radius_m)
    |   movel([0.589156, -1.411947, -2.554518, -0.745924, 1.570796, 2.159953],accel_mss,speed_ms,0,blend_radius_m)
    |   movel([0.588161, -1.416200, -2.551315, -0.744875, 1.570796, 2.158957],accel_mss,speed_ms,0,blend_radius_m)
    |   movel([0.587799, -1.417025, -2.550690, -0.744674, 1.570796, 2.158595],accel_mss,speed_ms,0,blend_radius_m)
    |   movel([0.587486, -1.417336, -2.550454, -0.744599, 1.570796, 2.158282],accel_mss,speed_ms,0,blend_radius_m)
    |   movel([0.587116, -1.417448, -2.550369, -0.744572, 1.570796, 2.157912],accel_mss,speed_ms,0,blend_radius_m)
    |   movel([0.586787, -1.417282, -2.550495, -0.744612, 1.570796, 2.157583],accel_mss,speed_ms,0,blend_radius_m)
    |   movel([0.586231, -1.416604, -2.551009, -0.744776, 1.570796, 2.157027],accel_mss,speed_ms,0,blend_radius_m)
    |   movel([0.585878, -1.415801, -2.551616, -0.744972, 1.570796, 2.156674],accel_mss,speed_ms,0,blend_radius_m)
    |   movel([0.585699, -1.414896, -2.552299, -0.745193, 1.570796, 2.156495],accel_mss,speed_ms,0,blend_radius_m)
    |   movel([0.585677, -1.413906, -2.553045, -0.745437, 1.570796, 2.156473],accel_mss,speed_ms,0,blend_radius_m)
    |   movel([0.586007, -1.411768, -2.554652, -0.745969, 1.570796, 2.156803],accel_mss,speed_ms,0,blend_radius_m)
    |   movel([0.586683, -1.409559, -2.556305, -0.746525, 1.570796, 2.157480],accel_mss,speed_ms,0,blend_radius_m)
    |   movel([0.584424, -1.413569, -2.553299, -0.745521, 1.570796, 2.155220],accel_mss,speed_ms,0,blend_radius_m)
    |   movel([0.583494, -1.415563, -2.551796, -0.745030, 1.570796, 2.154290],accel_mss,speed_ms,0,blend_radius_m)
    |   movel([0.582805, -1.417562, -2.550283, -0.744544, 1.570796, 2.153601],accel_mss,speed_ms,0,blend_radius_m)
    |   movel([0.582532, -1.419260, -2.548993, -0.744136, 1.570796, 2.153328],accel_mss,speed_ms,0,blend_radius_m)
    |   movel([0.582490, -1.422386, -2.546606, -0.743397, 1.570796, 2.153286],accel_mss,speed_ms,0,blend_radius_m)
    |   movel([0.582207, -1.424030, -2.545345, -0.743014, 1.570796, 2.153004],accel_mss,speed_ms,0,blend_radius_m)
    |   movel([0.582086, -1.424369, -2.545085, -0.742935, 1.570796, 2.152883],accel_mss,speed_ms,0,blend_radius_m)
    |   movel([0.581854, -1.424681, -2.544845, -0.742863, 1.570796, 2.152650],accel_mss,speed_ms,0,blend_radius_m)
    |   movel([0.581493, -1.424854, -2.544712, -0.742823, 1.570796, 2.152289],accel_mss,speed_ms,0,blend_radius_m)
    |   movel([0.581028, -1.424852, -2.544713, -0.742824, 1.570796, 2.151824],accel_mss,speed_ms,0,blend_radius_m)
    |   movel([0.579948, -1.424500, -2.544984, -0.742905, 1.570796, 2.150744],accel_mss,speed_ms,0,blend_radius_m)
    |   movel([0.578329, -1.423569, -2.545699, -0.743121, 1.570796, 2.149126],accel_mss,speed_ms,0,blend_radius_m)
    |   movel([0.577960, -1.424862, -2.544706, -0.742821, 1.570796, 2.148756],accel_mss,speed_ms,0,blend_radius_m)
    |   movel([0.577645, -1.426357, -2.543554, -0.742478, 1.570796, 2.148441],accel_mss,speed_ms,0,blend_radius_m)
    |   movel([0.577453, -1.428005, -2.542280, -0.742104, 1.570796, 2.148249],accel_mss,speed_ms,0,blend_radius_m)
    |   movel([0.577452, -1.429760, -2.540919, -0.741710, 1.570796, 2.148248],accel_mss,speed_ms,0,blend_radius_m)
    |   movel([0.578459, -1.432834, -2.538523, -0.741032, 1.570796, 2.149255],accel_mss,speed_ms,0,blend_radius_m)
    |   movel([0.578981, -1.434604, -2.537138, -0.740648, 1.570796, 2.149777],accel_mss,speed_ms,0,blend_radius_m)
    |   movel([0.579054, -1.435266, -2.536618, -0.740505, 1.570796, 2.149851],accel_mss,speed_ms,0,blend_radius_m)
    |   movel([0.578930, -1.435676, -2.536296, -0.740417, 1.570796, 2.149726],accel_mss,speed_ms,0,blend_radius_m)
    |   movel([0.578610, -1.435930, -2.536097, -0.740363, 1.570796, 2.149406],accel_mss,speed_ms,0,blend_radius_m)
    |   movel([0.578244, -1.436091, -2.535970, -0.740328, 1.570796, 2.149040],accel_mss,speed_ms,0,blend_radius_m)
    |   movel([0.577528, -1.436139, -2.535932, -0.740318, 1.570796, 2.148324],accel_mss,speed_ms,0,blend_radius_m)
    |   movel([0.577053, -1.435949, -2.536081, -0.740359, 1.570796, 2.147850],accel_mss,speed_ms,0,blend_radius_m)
    |   movel([0.576639, -1.435645, -2.536321, -0.740424, 1.570796, 2.147435],accel_mss,speed_ms,0,blend_radius_m)
    |   movel([0.575903, -1.434975, -2.536847, -0.740568, 1.570796, 2.146700],accel_mss,speed_ms,0,blend_radius_m)
    |   movel([0.575457, -1.436740, -2.535459, -0.740190, 1.570796, 2.146253],accel_mss,speed_ms,0,blend_radius_m)
    |   movel([0.575152, -1.438476, -2.534090, -0.739824, 1.570796, 2.145948],accel_mss,speed_ms,0,blend_radius_m)
    |   movel([0.574992, -1.440172, -2.532747, -0.739470, 1.570796, 2.145788],accel_mss,speed_ms,0,blend_radius_m)
    |   movel([0.574969, -1.441823, -2.531436, -0.739130, 1.570796, 2.145765],accel_mss,speed_ms,0,blend_radius_m)
    |   movel([0.575168, -1.443368, -2.530206, -0.738815, 1.570796, 2.145964],accel_mss,speed_ms,0,blend_radius_m)
    |   movel([0.575609, -1.444795, -2.529066, -0.738528, 1.570796, 2.146405],accel_mss,speed_ms,0,blend_radius_m)
    |   movel([0.576832, -1.447452, -2.526935, -0.738002, 1.570796, 2.147628],accel_mss,speed_ms,0,blend_radius_m)
    |   movel([0.577055, -1.448296, -2.526256, -0.737837, 1.570796, 2.147851],accel_mss,speed_ms,0,blend_radius_m)
    |   movel([0.576965, -1.448753, -2.525888, -0.737748, 1.570796, 2.147761],accel_mss,speed_ms,0,blend_radius_m)
    |   movel([0.576654, -1.449187, -2.525538, -0.737664, 1.570796, 2.147450],accel_mss,speed_ms,0,blend_radius_m)
    |   movel([0.576237, -1.449464, -2.525315, -0.737610, 1.570796, 2.147034],accel_mss,speed_ms,0,blend_radius_m)
    |   movel([0.575782, -1.449602, -2.525204, -0.737584, 1.570796, 2.146578],accel_mss,speed_ms,0,blend_radius_m)
    |   movel([0.574884, -1.449595, -2.525209, -0.737585, 1.570796, 2.145680],accel_mss,speed_ms,0,blend_radius_m)
    |   movel([0.573821, -1.449344, -2.525411, -0.737633, 1.570796, 2.144617],accel_mss,speed_ms,0,blend_radius_m)
    |   movel([0.572869, -1.448961, -2.525721, -0.737708, 1.570796, 2.143665],accel_mss,speed_ms,0,blend_radius_m)
    |   movel([0.572013, -1.448465, -2.526120, -0.737804, 1.570796, 2.142809],accel_mss,speed_ms,0,blend_radius_m)
    |   movel([0.571243, -1.447873, -2.526597, -0.737919, 1.570796, 2.142039],accel_mss,speed_ms,0,blend_radius_m)
    |   movel([0.571156, -1.449345, -2.525410, -0.737633, 1.570796, 2.141952],accel_mss,speed_ms,0,blend_radius_m)
    |   movel([0.571249, -1.450744, -2.524280, -0.737365, 1.570796, 2.142045],accel_mss,speed_ms,0,blend_radius_m)
    |   movel([0.571531, -1.452045, -2.523227, -0.737117, 1.570796, 2.142327],accel_mss,speed_ms,0,blend_radius_m)
    |   movel([0.572008, -1.453226, -2.522267, -0.736895, 1.570796, 2.142804],accel_mss,speed_ms,0,blend_radius_m)
    |   movel([0.572690, -1.454268, -2.521420, -0.736701, 1.570796, 2.143486],accel_mss,speed_ms,0,blend_radius_m)
    |   movel([0.573586, -1.455151, -2.520700, -0.736538, 1.570796, 2.144382],accel_mss,speed_ms,0,blend_radius_m)
    |   movel([0.574704, -1.455850, -2.520130, -0.736410, 1.570796, 2.145500],accel_mss,speed_ms,0,blend_radius_m)
    |   movel([0.576054, -1.456348, -2.519722, -0.736318, 1.570796, 2.146850],accel_mss,speed_ms,0,blend_radius_m)
    |   speed_ms = 0.005
    |   movel([0.576054, -1.448109, -2.516058, -0.748222, 1.570796, 2.146850],accel_mss,speed_ms,0,blend_radius_m)
    |   speed_ms = 0.040
    |   movel([0.585604, -1.442287, -2.520731, -0.749370, 1.570796, 2.156400],accel_mss,speed_ms,0,blend_radius_m)
    |   speed_ms = 0.005
    |   movel([0.585604, -1.450572, -2.524420, -0.737398, 1.570796, 2.156400],accel_mss,speed_ms,0,blend_radius_m)
    |   speed_ms = 0.025
    |   movel([0.583814, -1.448240, -2.526302, -0.737848, 1.570796, 2.154611],accel_mss,speed_ms,0,blend_radius_m)
    |   movel([0.583126, -1.447097, -2.527220, -0.738071, 1.570796, 2.153922],accel_mss,speed_ms,0,blend_radius_m)
    |   movel([0.582592, -1.445916, -2.528168, -0.738305, 1.570796, 2.153389],accel_mss,speed_ms,0,blend_radius_m)
    |   movel([0.582226, -1.444649, -2.529183, -0.738557, 1.570796, 2.153022],accel_mss,speed_ms,0,blend_radius_m)
    |   movel([0.582039, -1.443255, -2.530296, -0.738838, 1.570796, 2.152835],accel_mss,speed_ms,0,blend_radius_m)
    |   movel([0.582043, -1.441690, -2.531542, -0.739157, 1.570796, 2.152839],accel_mss,speed_ms,0,blend_radius_m)
    |   movel([0.582253, -1.439911, -2.532954, -0.739524, 1.570796, 2.153050],accel_mss,speed_ms,0,blend_radius_m)
    |   movel([0.583077, -1.436109, -2.535956, -0.740325, 1.570796, 2.153873],accel_mss,speed_ms,0,blend_radius_m)
    |   movel([0.584263, -1.432233, -2.538993, -0.741163, 1.570796, 2.155059],accel_mss,speed_ms,0,blend_radius_m)
    |   movel([0.585769, -1.428306, -2.542047, -0.742036, 1.570796, 2.156566],accel_mss,speed_ms,0,blend_radius_m)
    |   movel([0.587548, -1.424355, -2.545096, -0.742938, 1.570796, 2.158344],accel_mss,speed_ms,0,blend_radius_m)
    |   movel([0.589196, -1.421115, -2.547579, -0.743696, 1.570796, 2.159993],accel_mss,speed_ms,0,blend_radius_m)
    |   movel([0.590996, -1.417874, -2.550046, -0.744469, 1.570796, 2.161792],accel_mss,speed_ms,0,blend_radius_m)
    |   movel([0.594940, -1.411377, -2.554946, -0.746067, 1.570796, 2.165736],accel_mss,speed_ms,0,blend_radius_m)
    |   movel([0.609438, -1.388730, -2.571533, -0.752125, 1.570796, 2.180234],accel_mss,speed_ms,0,blend_radius_m)
    |   movel([0.612520, -1.383868, -2.574997, -0.753524, 1.570796, 2.183317],accel_mss,speed_ms,0,blend_radius_m)
    |   movel([0.615548, -1.378943, -2.578470, -0.754976, 1.570796, 2.186344],accel_mss,speed_ms,0,blend_radius_m)
    |   movel([0.618446, -1.373967, -2.581944, -0.756479, 1.570796, 2.189243],accel_mss,speed_ms,0,blend_radius_m)
    |   movel([0.621146, -1.368941, -2.585416, -0.758032, 1.570796, 2.191942],accel_mss,speed_ms,0,blend_radius_m)
    |   movel([0.623574, -1.363874, -2.588880, -0.759635, 1.570796, 2.194371],accel_mss,speed_ms,0,blend_radius_m)
    |   movel([0.625657, -1.358775, -2.592330, -0.761284, 1.570796, 2.196453],accel_mss,speed_ms,0,blend_radius_m)
    |   movel([0.626927, -1.355048, -2.594828, -0.762513, 1.570796, 2.197723],accel_mss,speed_ms,0,blend_radius_m)
    |   movel([0.628014, -1.351222, -2.597372, -0.763795, 1.570796, 2.198811],accel_mss,speed_ms,0,blend_radius_m)
    |   movel([0.628873, -1.347360, -2.599920, -0.765109, 1.570796, 2.199669],accel_mss,speed_ms,0,blend_radius_m)
    |   movel([0.629455, -1.343522, -2.602432, -0.766436, 1.570796, 2.200252],accel_mss,speed_ms,0,blend_radius_m)
    |   movel([0.629717, -1.339772, -2.604866, -0.767752, 1.570796, 2.200513],accel_mss,speed_ms,0,blend_radius_m)
    |   movel([0.629612, -1.336173, -2.607183, -0.769033, 1.570796, 2.200408],accel_mss,speed_ms,0,blend_radius_m)
    |   movel([0.629087, -1.332796, -2.609342, -0.770251, 1.570796, 2.199883],accel_mss,speed_ms,0,blend_radius_m)
    |   movel([0.628098, -1.329712, -2.611300, -0.771377, 1.570796, 2.198895],accel_mss,speed_ms,0,blend_radius_m)
    |   movel([0.627440, -1.328399, -2.612130, -0.771860, 1.570796, 2.198236],accel_mss,speed_ms,0,blend_radius_m)
    |   movel([0.626623, -1.327191, -2.612891, -0.772307, 1.570796, 2.197419],accel_mss,speed_ms,0,blend_radius_m)
    |   movel([0.625646, -1.326111, -2.613570, -0.772708, 1.570796, 2.196443],accel_mss,speed_ms,0,blend_radius_m)
    |   movel([0.624512, -1.325183, -2.614152, -0.773054, 1.570796, 2.195308],accel_mss,speed_ms,0,blend_radius_m)
    |   movel([0.623225, -1.324426, -2.614626, -0.773337, 1.570796, 2.194021],accel_mss,speed_ms,0,blend_radius_m)
    |   movel([0.621781, -1.323866, -2.614976, -0.773547, 1.570796, 2.192578],accel_mss,speed_ms,0,blend_radius_m)
    |   movel([0.620189, -1.323521, -2.615192, -0.773676, 1.570796, 2.190985],accel_mss,speed_ms,0,blend_radius_m)
    |   movel([0.618447, -1.323417, -2.615256, -0.773715, 1.570796, 2.189243],accel_mss,speed_ms,0,blend_radius_m)
    |   speed_ms = 0.005
    |   movel([0.618447, -1.314215, -2.611012, -0.787163, 1.570796, 2.189243],accel_mss,speed_ms,0,blend_radius_m)
    |   speed_ms = 0.040
    |   movel([0.619533, -1.300841, -2.619131, -0.792417, 1.570796, 2.190329],accel_mss,speed_ms,0,blend_radius_m)
    |   speed_ms = 0.005
    |   movel([0.619533, -1.310126, -2.623436, -0.778827, 1.570796, 2.190329],accel_mss,speed_ms,0,blend_radius_m)
    |   speed_ms = 0.025
    |   movel([0.620109, -1.308679, -2.624312, -0.779398, 1.570796, 2.190905],accel_mss,speed_ms,0,blend_radius_m)
    |   movel([0.620827, -1.307239, -2.625181, -0.779968, 1.570796, 2.191624],accel_mss,speed_ms,0,blend_radius_m)
    |   movel([0.622599, -1.304391, -2.626893, -0.781105, 1.570796, 2.193395],accel_mss,speed_ms,0,blend_radius_m)
    |   movel([0.624684, -1.301583, -2.628570, -0.782236, 1.570796, 2.195480],accel_mss,speed_ms,0,blend_radius_m)
    |   movel([0.626909, -1.298827, -2.630206, -0.783356, 1.570796, 2.197705],accel_mss,speed_ms,0,blend_radius_m)
    |   speed_ms = 0.005
    |   movel([0.626909, -1.289474, -2.625850, -0.797065, 1.570796, 2.197705],accel_mss,speed_ms,0,blend_radius_m)
    |   speed_ms = 0.040
    |   movel([0.629236, -1.292240, -2.624231, -0.795919, 1.570796, 2.200032],accel_mss,speed_ms,0,blend_radius_m)
    |   speed_ms = 0.005
    |   movel([0.629236, -1.301576, -2.628574, -0.782239, 1.570796, 2.200032],accel_mss,speed_ms,0,blend_radius_m)
    |   speed_ms = 0.025
    |   movel([0.629448, -1.300276, -2.629348, -0.782766, 1.570796, 2.200244],accel_mss,speed_ms,0,blend_radius_m)
    |   movel([0.629802, -1.298978, -2.630117, -0.783294, 1.570796, 2.200598],accel_mss,speed_ms,0,blend_radius_m)
    |   movel([0.630897, -1.296389, -2.631645, -0.784355, 1.570796, 2.201693],accel_mss,speed_ms,0,blend_radius_m)
    |   movel([0.632440, -1.293836, -2.633144, -0.785409, 1.570796, 2.203236],accel_mss,speed_ms,0,blend_radius_m)
    |   movel([0.634351, -1.291335, -2.634604, -0.786450, 1.570796, 2.205148],accel_mss,speed_ms,0,blend_radius_m)
    |   movel([0.636548, -1.288908, -2.636013, -0.787468, 1.570796, 2.207344],accel_mss,speed_ms,0,blend_radius_m)
    |   movel([0.638945, -1.286578, -2.637359, -0.788452, 1.570796, 2.209741],accel_mss,speed_ms,0,blend_radius_m)
    |   movel([0.641458, -1.284365, -2.638630, -0.789393, 1.570796, 2.212255],accel_mss,speed_ms,0,blend_radius_m)
    |   movel([0.644002, -1.282293, -2.639816, -0.790280, 1.570796, 2.214798],accel_mss,speed_ms,0,blend_radius_m)
    |   speed_ms = 0.005
    |   movel([0.644002, -1.272846, -2.635384, -0.804159, 1.570796, 2.214798],accel_mss,speed_ms,0,blend_radius_m)
    |   speed_ms = 0.040
    |   movel([0.669072, -1.259735, -2.642660, -0.809994, 1.570796, 2.239868],accel_mss,speed_ms,0,blend_radius_m)
    |   speed_ms = 0.005
    |   movel([0.669072, -1.269252, -2.647151, -0.795986, 1.570796, 2.239868],accel_mss,speed_ms,0,blend_radius_m)
    |   speed_ms = 0.025
    |   movel([0.666960, -1.269846, -2.646821, -0.795721, 1.570796, 2.237757],accel_mss,speed_ms,0,blend_radius_m)
    |   movel([0.664756, -1.270617, -2.646393, -0.795379, 1.570796, 2.235552],accel_mss,speed_ms,0,blend_radius_m)
    |   movel([0.662493, -1.271553, -2.645872, -0.794964, 1.570796, 2.233289],accel_mss,speed_ms,0,blend_radius_m)
    |   movel([0.660197, -1.272645, -2.645263, -0.794481, 1.570796, 2.230993],accel_mss,speed_ms,0,blend_radius_m)
    |   movel([0.657902, -1.273885, -2.644570, -0.793935, 1.570796, 2.228698],accel_mss,speed_ms,0,blend_radius_m)
    |   movel([0.655639, -1.275258, -2.643799, -0.793332, 1.570796, 2.226436],accel_mss,speed_ms,0,blend_radius_m)
    |   movel([0.653438, -1.276760, -2.642954, -0.792675, 1.570796, 2.224235],accel_mss,speed_ms,0,blend_radius_m)
    |   movel([0.651329, -1.278380, -2.642039, -0.791970, 1.570796, 2.222125],accel_mss,speed_ms,0,blend_radius_m)
    |   movel([0.649343, -1.280103, -2.641063, -0.791223, 1.570796, 2.220140],accel_mss,speed_ms,0,blend_radius_m)
    |   movel([0.647509, -1.281924, -2.640026, -0.790439, 1.570796, 2.218305],accel_mss,speed_ms,0,blend_radius_m)
    |   movel([0.645855, -1.283830, -2.638937, -0.789622, 1.570796, 2.216652],accel_mss,speed_ms,0,blend_radius_m)
    |   movel([0.644412, -1.285811, -2.637800, -0.788778, 1.570796, 2.215208],accel_mss,speed_ms,0,blend_radius_m)
    |   movel([0.643209, -1.287858, -2.636620, -0.787911, 1.570796, 2.214005],accel_mss,speed_ms,0,blend_radius_m)
    |   movel([0.642274, -1.289961, -2.635403, -0.787025, 1.570796, 2.213070],accel_mss,speed_ms,0,blend_radius_m)
    |   movel([0.641632, -1.292110, -2.634152, -0.786127, 1.570796, 2.212428],accel_mss,speed_ms,0,blend_radius_m)
    |   movel([0.641312, -1.294297, -2.632874, -0.785218, 1.570796, 2.212108],accel_mss,speed_ms,0,blend_radius_m)
    |   speed_ms = 0.005
    |   movel([0.641312, -1.284918, -2.628497, -0.798974, 1.570796, 2.212108],accel_mss,speed_ms,0,blend_radius_m)
    |   speed_ms = 0.040
    |   movel([0.651214, -1.282509, -2.629886, -0.799994, 1.570796, 2.222010],accel_mss,speed_ms,0,blend_radius_m)
    |   speed_ms = 0.005
    |   movel([0.651214, -1.291902, -2.634274, -0.786213, 1.570796, 2.222010],accel_mss,speed_ms,0,blend_radius_m)
    |   speed_ms = 0.025
    |   movel([0.651897, -1.290182, -2.635274, -0.786933, 1.570796, 2.222693],accel_mss,speed_ms,0,blend_radius_m)
    |   movel([0.652726, -1.288451, -2.636278, -0.787660, 1.570796, 2.223522],accel_mss,speed_ms,0,blend_radius_m)
    |   movel([0.653690, -1.286727, -2.637273, -0.788389, 1.570796, 2.224486],accel_mss,speed_ms,0,blend_radius_m)
    |   movel([0.654782, -1.285021, -2.638254, -0.789114, 1.570796, 2.225579],accel_mss,speed_ms,0,blend_radius_m)
    |   movel([0.655991, -1.283349, -2.639213, -0.789828, 1.570796, 2.226787],accel_mss,speed_ms,0,blend_radius_m)
    |   movel([0.657310, -1.281724, -2.640140, -0.790525, 1.570796, 2.228106],accel_mss,speed_ms,0,blend_radius_m)
    |   movel([0.658732, -1.280158, -2.641031, -0.791200, 1.570796, 2.229528],accel_mss,speed_ms,0,blend_radius_m)
    |   movel([0.660243, -1.278670, -2.641875, -0.791844, 1.570796, 2.231039],accel_mss,speed_ms,0,blend_radius_m)
    |   movel([0.661835, -1.277271, -2.642666, -0.792452, 1.570796, 2.232631],accel_mss,speed_ms,0,blend_radius_m)
    |   movel([0.663502, -1.275977, -2.643395, -0.793017, 1.570796, 2.234299],accel_mss,speed_ms,0,blend_radius_m)
    |   movel([0.665227, -1.274805, -2.644054, -0.793530, 1.570796, 2.236023],accel_mss,speed_ms,0,blend_radius_m)
    |   movel([0.667007, -1.273766, -2.644636, -0.793987, 1.570796, 2.237804],accel_mss,speed_ms,0,blend_radius_m)
    |   movel([0.668830, -1.272877, -2.645133, -0.794378, 1.570796, 2.239626],accel_mss,speed_ms,0,blend_radius_m)
    |   movel([0.670684, -1.272153, -2.645538, -0.794698, 1.570796, 2.241481],accel_mss,speed_ms,0,blend_radius_m)
    |   movel([0.672560, -1.271611, -2.645840, -0.794938, 1.570796, 2.243356],accel_mss,speed_ms,0,blend_radius_m)
    |   movel([0.674444, -1.271261, -2.646035, -0.795093, 1.570796, 2.245241],accel_mss,speed_ms,0,blend_radius_m)
    |   movel([0.676214, -1.271136, -2.646104, -0.795149, 1.570796, 2.247010],accel_mss,speed_ms,0,blend_radius_m)
    |   movel([0.677859, -1.271228, -2.646053, -0.795108, 1.570796, 2.248656],accel_mss,speed_ms,0,blend_radius_m)
    |   movel([0.679377, -1.271521, -2.645890, -0.794978, 1.570796, 2.250174],accel_mss,speed_ms,0,blend_radius_m)
    |   movel([0.680769, -1.272004, -2.645621, -0.794764, 1.570796, 2.251565],accel_mss,speed_ms,0,blend_radius_m)
    |   movel([0.682031, -1.272660, -2.645254, -0.794474, 1.570796, 2.252827],accel_mss,speed_ms,0,blend_radius_m)
    |   movel([0.683157, -1.273479, -2.644797, -0.794113, 1.570796, 2.253954],accel_mss,speed_ms,0,blend_radius_m)
    |   movel([0.684155, -1.274441, -2.644258, -0.793690, 1.570796, 2.254951],accel_mss,speed_ms,0,blend_radius_m)
    |   movel([0.685014, -1.275535, -2.643644, -0.793211, 1.570796, 2.255810],accel_mss,speed_ms,0,blend_radius_m)
    |   movel([0.685737, -1.276745, -2.642962, -0.792681, 1.570796, 2.256533],accel_mss,speed_ms,0,blend_radius_m)
    |   movel([0.686774, -1.279456, -2.641430, -0.791503, 1.570796, 2.257571],accel_mss,speed_ms,0,blend_radius_m)
    |   movel([0.687082, -1.280926, -2.640595, -0.790868, 1.570796, 2.257879],accel_mss,speed_ms,0,blend_radius_m)
    |   movel([0.687283, -1.284028, -2.638824, -0.789537, 1.570796, 2.258079],accel_mss,speed_ms,0,blend_radius_m)
    |   movel([0.687174, -1.285630, -2.637905, -0.788855, 1.570796, 2.257970],accel_mss,speed_ms,0,blend_radius_m)
    |   movel([0.686921, -1.287246, -2.636973, -0.788169, 1.570796, 2.257718],accel_mss,speed_ms,0,blend_radius_m)
    |   speed_ms = 0.005
